LIN {X 0.073,Y -492.904,Z 865.526,A 0.000,B 0.000,C 90.000,E1 274.645} C_DIS
LIN {X -0.220,Y -493.120,Z 865.523,A 0.000,B 0.000,C 90.000,E1 274.188} C_DIS
LIN {X 0.017,Y -492.879,Z 865.520,A 0.000,B 0.000,C 90.000,E1 273.669} C_DIS
LIN {X 0.225,Y -492.231,Z 865.518,A 0.000,B 0.000,C 90.000,E1 273.154} C_DIS
LIN {X -0.033,Y -491.091,Z 865.515,A 0.000,B 0.000,C 90.000,E1 272.694} C_DIS
LIN {X 0.172,Y -489.509,Z 865.512,A 0.000,B 0.000,C 90.000,E1 272.178} C_DIS
LIN {X -0.101,Y -487.367,Z 865.509,A 0.000,B 0.000,C 90.000,E1 271.718} C_DIS
LIN {X 0.088,Y -484.709,Z 865.507,A 0.000,B 0.000,C 90.000,E1 271.203} C_DIS
LIN {X -0.225,Y -481.334,Z 865.504,A 0.000,B 0.000,C 90.000,E1 270.745} C_DIS
LIN {X -0.070,Y -477.260,Z 865.501,A 0.000,B 0.000,C 90.000,E1 270.229} C_DIS
LIN {X 0.060,Y -472.369,Z 865.498,A 0.000,B 0.000,C 90.000,E1 269.714} C_DIS
LIN {X -0.155,Y -466.565,Z 865.496,A 0.000,B 0.000,C 90.000,E1 269.255} C_DIS
LIN {X 0.090,Y -460.380,Z 865.493,A 0.000,B 0.000,C 90.000,E1 268.797} C_DIS
LIN {X -0.019,Y -457.282,Z 865.492,A 0.000,B 0.000,C 90.000,E1 268.625} C_DIS
LIN {X 0.043,Y -450.188,Z 865.490,A 0.000,B 0.000,C 90.000,E1 268.282} C_DIS
LIN {X 0.171,Y -442.949,Z 865.489,A 0.000,B 0.000,C 90.000,E1 267.993} C_DIS
LIN {X -0.152,Y -435.156,Z 865.488,A 0.000,B 0.000,C 90.000,E1 267.822} C_DIS
LIN {X -0.075,Y -427.085,Z 865.487,A 0.000,B 0.000,C 90.000,E1 267.650} C_DIS
LIN {X -0.084,Y -416.791,Z 865.486,A 0.000,B 0.000,C 90.000,E1 267.535} C_DIS
LIN {X 0.160,Y -410.055,Z 865.486,A 0.000,B 0.000,C 90.000,E1 267.478} C_DIS
LIN {X 0.053,Y -181.050,Z 865.486,A 0.000,B 0.000,C 90.000,E1 267.478} C_DIS
LIN {X -0.048,Y -180.907,Z 865.475,A 0.000,B 0.000,C 90.000,E1 265.469} C_DIS
LIN {X 0.008,Y -180.730,Z 865.470,A 0.000,B 0.000,C 90.000,E1 264.609} C_DIS
LIN {X -0.070,Y -178.819,Z 865.442,A 0.000,B 0.000,C 90.000,E1 259.567} C_DIS
LIN {X 0.012,Y -175.863,Z 865.414,A 0.000,B 0.000,C 90.000,E1 254.448} C_DIS
LIN {X 0.061,Y -173.830,Z 865.399,A 0.000,B 0.000,C 90.000,E1 251.873} C_DIS
LIN {X -0.004,Y -171.497,Z 865.380,A 0.000,B 0.000,C 90.000,E1 248.465} C_DIS
LIN {X -0.017,Y -167.726,Z 865.356,A 0.000,B 0.000,C 90.000,E1 244.152} C_DIS
LIN {X -0.001,Y -166.421,Z 865.347,A 0.000,B 0.000,C 90.000,E1 242.410} C_DIS
LIN {X -0.002,Y -163.142,Z 865.327,A 0.000,B 0.000,C 90.000,E1 238.918} C_DIS
LIN {X -0.037,Y -161.096,Z 865.313,A 0.000,B 0.000,C 90.000,E1 236.294} C_DIS
LIN {X -0.053,Y -157.825,Z 865.293,A 0.000,B 0.000,C 90.000,E1 232.763} C_DIS
LIN {X 0.010,Y -155.859,Z 865.278,A 0.000,B 0.000,C 90.000,E1 230.070} C_DIS
LIN {X 0.066,Y -152.109,Z 865.253,A 0.000,B 0.000,C 90.000,E1 225.567} C_DIS
LIN {X -0.026,Y -150.359,Z 865.238,A 0.000,B 0.000,C 90.000,E1 222.894} C_DIS
LIN {X 0.013,Y -147.095,Z 865.213,A 0.000,B 0.000,C 90.000,E1 218.338} C_DIS
LIN {X 0.008,Y -145.665,Z 865.198,A 0.000,B 0.000,C 90.000,E1 215.598} C_DIS
LIN {X 0.010,Y -143.047,Z 865.172,A 0.000,B 0.000,C 90.000,E1 211.003} C_DIS
LIN {X 0.011,Y -141.671,Z 865.152,A 0.000,B 0.000,C 90.000,E1 207.308} C_DIS
LIN {X 0.055,Y -139.452,Z 865.116,A 0.000,B 0.000,C 90.000,E1 200.791} C_DIS
LIN {X -0.023,Y -139.186,Z 865.105,A 0.000,B 0.000,C 90.000,E1 198.960} C_DIS
LIN {X -0.001,Y -138.322,Z 865.053,A 0.000,B 0.000,C 90.000,E1 189.613} C_DIS
LIN {X 0.006,Y -139.460,Z 865.007,A 0.000,B 0.000,C 90.000,E1 181.203} C_DIS
LIN {X -0.054,Y -141.016,Z 864.976,A 0.000,B 0.000,C 90.000,E1 175.641} C_DIS
LIN {X 0.037,Y -142.770,Z 864.955,A 0.000,B 0.000,C 90.000,E1 171.894} C_DIS
LIN {X -0.008,Y -145.180,Z 864.929,A 0.000,B 0.000,C 90.000,E1 167.297} C_DIS
LIN {X 0.025,Y -147.803,Z 864.909,A 0.000,B 0.000,C 90.000,E1 163.614} C_DIS
LIN {X -0.080,Y -150.489,Z 864.889,A 0.000,B 0.000,C 90.000,E1 160.007} C_DIS
LIN {X -0.007,Y -153.944,Z 864.869,A 0.000,B 0.000,C 90.000,E1 156.357} C_DIS
LIN {X 0.056,Y -157.356,Z 864.849,A 0.000,B 0.000,C 90.000,E1 152.743} C_DIS
LIN {X -0.001,Y -161.552,Z 864.829,A 0.000,B 0.000,C 90.000,E1 149.203} C_DIS
LIN {X 0.011,Y -165.749,Z 864.809,A 0.000,B 0.000,C 90.000,E1 145.674} C_DIS
LIN {X -0.002,Y -170.704,Z 864.790,A 0.000,B 0.000,C 90.000,E1 142.190} C_DIS
LIN {X -0.090,Y -175.578,Z 864.771,A 0.000,B 0.000,C 90.000,E1 138.771} C_DIS
LIN {X 0.029,Y -181.196,Z 864.752,A 0.000,B 0.000,C 90.000,E1 135.324} C_DIS
LIN {X 0.022,Y -186.657,Z 864.733,A 0.000,B 0.000,C 90.000,E1 131.962} C_DIS
LIN {X -0.034,Y -191.262,Z 864.719,A 0.000,B 0.000,C 90.000,E1 129.483} C_DIS
LIN {X -0.025,Y -193.092,Z 864.713,A 0.000,B 0.000,C 90.000,E1 128.382} C_DIS
LIN {X -0.072,Y -294.130,Z 864.713,A 0.000,B 0.000,C 90.000,E1 128.382} C_DIS
LIN {X 0.045,Y -296.837,Z 864.713,A 0.000,B 0.000,C 90.000,E1 128.302} C_DIS
LIN {X -0.152,Y -301.150,Z 864.711,A 0.000,B 0.000,C 90.000,E1 128.096} C_DIS
LIN {X 0.072,Y -303.688,Z 864.710,A 0.000,B 0.000,C 90.000,E1 127.810} C_DIS
LIN {X -0.038,Y -307.442,Z 864.707,A 0.000,B 0.000,C 90.000,E1 127.282} C_DIS
LIN {X -0.019,Y -309.008,Z 864.705,A 0.000,B 0.000,C 90.000,E1 126.950} C_DIS
LIN {X 0.186,Y -310.237,Z 864.703,A 0.000,B 0.000,C 90.000,E1 126.583} C_DIS
LIN {X -0.127,Y -321.379,Z 864.684,A 0.000,B 0.000,C 90.000,E1 123.086} C_DIS
LIN {X 0.019,Y -331.855,Z 864.668,A 0.000,B 0.000,C 90.000,E1 120.207} C_DIS
LIN {X 0.149,Y -343.684,Z 864.652,A 0.000,B 0.000,C 90.000,E1 117.385} C_DIS
LIN {X 0.142,Y -356.977,Z 864.637,A 0.000,B 0.000,C 90.000,E1 114.643} C_DIS
LIN {X -0.014,Y -370.114,Z 864.624,A 0.000,B 0.000,C 90.000,E1 112.280} C_DIS
LIN {X 0.019,Y -384.590,Z 864.611,A 0.000,B 0.000,C 90.000,E1 109.939} C_DIS
LIN {X 0.152,Y -400.512,Z 864.598,A 0.000,B 0.000,C 90.000,E1 107.638} C_DIS
LIN {X 0.055,Y -417.992,Z 864.586,A 0.000,B 0.000,C 90.000,E1 105.426} C_DIS
LIN {X -0.238,Y -437.140,Z 864.574,A 0.000,B 0.000,C 90.000,E1 103.300} C_DIS
LIN {X 0.008,Y -457.271,Z 864.562,A 0.000,B 0.000,C 90.000,E1 101.243} C_DIS
LIN {X -0.124,Y -467.492,Z 864.557,A 0.000,B 0.000,C 90.000,E1 100.310} C_DIS
LIN {X -0.128,Y -469.515,Z 864.556,A 0.000,B 0.000,C 90.000,E1 100.074} C_DIS
LIN {X -0.214,Y -471.052,Z 864.555,A 0.000,B 0.000,C 90.000,E1 99.849} C_DIS
LIN {X 0.105,Y -472.304,Z 864.553,A 0.000,B 0.000,C 90.000,E1 99.557} C_DIS
LIN {X -0.042,Y -473.223,Z 864.552,A 0.000,B 0.000,C 90.000,E1 99.321} C_DIS
LIN {X 0.070,Y -474.227,Z 864.549,A 0.000,B 0.000,C 90.000,E1 98.803} C_DIS
LIN {X 0.259,Y -474.248,Z 864.546,A 0.000,B 0.000,C 90.000,E1 98.276} C_DIS
LIN {X -0.087,Y -473.293,Z 864.543,A 0.000,B 0.000,C 90.000,E1 97.814} C_DIS
LIN {X 0.039,Y -471.201,Z 864.541,A 0.000,B 0.000,C 90.000,E1 97.296} C_DIS
LIN {X 0.195,Y -453.697,Z 864.525,A 0.000,B 0.000,C 90.000,E1 94.473} C_DIS
LIN {X -0.110,Y -443.186,Z 864.515,A 0.000,B 0.000,C 90.000,E1 92.694} C_DIS
LIN {X 0.075,Y -433.849,Z 864.506,A 0.000,B 0.000,C 90.000,E1 91.088} C_DIS
LIN {X 0.086,Y -424.216,Z 864.497,A 0.000,B 0.000,C 90.000,E1 89.484} C_DIS
LIN {X 0.030,Y -412.818,Z 864.487,A 0.000,B 0.000,C 90.000,E1 87.593} C_DIS
LIN {X 0.175,Y -401.391,Z 864.476,A 0.000,B 0.000,C 90.000,E1 85.641} C_DIS
LIN {X 0.157,Y -388.423,Z 864.463,A 0.000,B 0.000,C 90.000,E1 83.394} C_DIS
LIN {X -0.115,Y -375.665,Z 864.451,A 0.000,B 0.000,C 90.000,E1 81.141} C_DIS
LIN {X 0.130,Y -361.540,Z 864.436,A 0.000,B 0.000,C 90.000,E1 78.465} C_DIS
LIN {X -0.089,Y -350.608,Z 864.424,A 0.000,B 0.000,C 90.000,E1 76.408} C_DIS
LIN {X -0.118,Y -338.191,Z 864.411,A 0.000,B 0.000,C 90.000,E1 73.976} C_DIS
LIN {X 0.060,Y -326.043,Z 864.397,A 0.000,B 0.000,C 90.000,E1 71.456} C_DIS
LIN {X 0.064,Y -312.889,Z 864.381,A 0.000,B 0.000,C 90.000,E1 68.592} C_DIS
LIN {X -0.133,Y -302.956,Z 864.369,A 0.000,B 0.000,C 90.000,E1 66.357} C_DIS
LIN {X -0.027,Y -291.711,Z 864.354,A 0.000,B 0.000,C 90.000,E1 63.691} C_DIS
LIN {X 0.089,Y -281.990,Z 864.341,A 0.000,B 0.000,C 90.000,E1 61.307} C_DIS
LIN {X -0.042,Y -271.106,Z 864.325,A 0.000,B 0.000,C 90.000,E1 58.584} C_DIS
LIN {X 0.015,Y -258.194,Z 864.306,A 0.000,B 0.000,C 90.000,E1 55.055} C_DIS
LIN {X -0.021,Y -247.643,Z 864.288,A 0.000,B 0.000,C 90.000,E1 51.823} C_DIS
LIN {X -0.068,Y -237.007,Z 864.267,A 0.000,B 0.000,C 90.000,E1 48.162} C_DIS
LIN {X 0.017,Y -227.185,Z 864.247,A 0.000,B 0.000,C 90.000,E1 44.393} C_DIS
LIN {X 0.128,Y -218.020,Z 864.225,A 0.000,B 0.000,C 90.000,E1 40.539} C_DIS
LIN {X 0.064,Y -211.123,Z 864.208,A 0.000,B 0.000,C 90.000,E1 37.443} C_DIS
LIN {X 0.021,Y -203.152,Z 864.186,A 0.000,B 0.000,C 90.000,E1 33.499} C_DIS
LIN {X 0.075,Y -195.967,Z 864.164,A 0.000,B 0.000,C 90.000,E1 29.461} C_DIS
LIN {X -0.043,Y -190.896,Z 864.146,A 0.000,B 0.000,C 90.000,E1 26.232} C_DIS
LIN {X 0.069,Y -186.582,Z 864.127,A 0.000,B 0.000,C 90.000,E1 22.898} C_DIS
LIN {X 0.079,Y -182.215,Z 864.104,A 0.000,B 0.000,C 90.000,E1 18.725} C_DIS
LIN {X 0.014,Y -178.992,Z 864.081,A 0.000,B 0.000,C 90.000,E1 14.537} C_DIS
LIN {X -0.068,Y -176.333,Z 864.048,A 0.000,B 0.000,C 90.000,E1 8.624} C_DIS
LIN {X -0.078,Y -177.590,Z 863.974,A 0.000,B 0.000,C 90.000,E1 355.298} C_DIS
LIN {X -0.075,Y -180.602,Z 863.945,A 0.000,B 0.000,C 90.000,E1 350.208} C_DIS
LIN {X -0.059,Y -184.287,Z 863.922,A 0.000,B 0.000,C 90.000,E1 345.992} C_DIS
LIN {X -0.063,Y -189.055,Z 863.899,A 0.000,B 0.000,C 90.000,E1 341.819} C_DIS
LIN {X 0.099,Y -193.603,Z 863.880,A 0.000,B 0.000,C 90.000,E1 338.465} C_DIS
LIN {X 0.005,Y -200.178,Z 863.858,A 0.000,B 0.000,C 90.000,E1 334.409} C_DIS
LIN {X 0.014,Y -207.406,Z 863.836,A 0.000,B 0.000,C 90.000,E1 330.383} C_DIS
LIN {X 0.024,Y -215.337,Z 863.813,A 0.000,B 0.000,C 90.000,E1 326.421} C_DIS
LIN {X 0.071,Y -222.281,Z 863.796,A 0.000,B 0.000,C 90.000,E1 323.290} C_DIS
LIN {X 0.113,Y -230.938,Z 863.777,A 0.000,B 0.000,C 90.000,E1 319.828} C_DIS
LIN {X 0.083,Y -239.422,Z 863.760,A 0.000,B 0.000,C 90.000,E1 316.824} C_DIS
LIN {X 0.087,Y -248.774,Z 863.744,A 0.000,B 0.000,C 90.000,E1 313.866} C_DIS
LIN {X 0.019,Y -260.312,Z 863.726,A 0.000,B 0.000,C 90.000,E1 310.620} C_DIS
LIN {X -0.022,Y -272.802,Z 863.708,A 0.000,B 0.000,C 90.000,E1 307.443} C_DIS
LIN {X 0.013,Y -286.471,Z 863.691,A 0.000,B 0.000,C 90.000,E1 304.326} C_DIS
LIN {X -0.201,Y -301.452,Z 863.674,A 0.000,B 0.000,C 90.000,E1 301.337} C_DIS
LIN {X 0.003,Y -314.127,Z 863.661,A 0.000,B 0.000,C 90.000,E1 298.999} C_DIS
LIN {X -0.044,Y -325.947,Z 863.650,A 0.000,B 0.000,C 90.000,E1 297.078} C_DIS
LIN {X -0.044,Y -345.450,Z 863.635,A 0.000,B 0.000,C 90.000,E1 294.259} C_DIS
LIN {X 0.034,Y -369.064,Z 863.618,A 0.000,B 0.000,C 90.000,E1 291.227} C_DIS
LIN {X 0.144,Y -394.598,Z 863.602,A 0.000,B 0.000,C 90.000,E1 288.362} C_DIS
LIN {X -0.033,Y -412.830,Z 863.592,A 0.000,B 0.000,C 90.000,E1 286.496} C_DIS
LIN {X 0.054,Y -422.816,Z 863.586,A 0.000,B 0.000,C 90.000,E1 285.426} C_DIS
LIN {X 0.035,Y -432.657,Z 863.580,A 0.000,B 0.000,C 90.000,E1 284.356} C_DIS
LIN {X -0.054,Y -442.279,Z 863.574,A 0.000,B 0.000,C 90.000,E1 283.300} C_DIS
LIN {X -0.026,Y -451.331,Z 863.568,A 0.000,B 0.000,C 90.000,E1 282.243} C_DIS
LIN {X 0.119,Y -459.815,Z 863.562,A 0.000,B 0.000,C 90.000,E1 281.186} C_DIS
LIN {X -0.189,Y -467.691,Z 863.557,A 0.000,B 0.000,C 90.000,E1 280.197} C_DIS
LIN {X 0.055,Y -474.900,Z 863.551,A 0.000,B 0.000,C 90.000,E1 279.151} C_DIS
LIN {X 0.045,Y -479.741,Z 863.547,A 0.000,B 0.000,C 90.000,E1 278.398} C_DIS
LIN {X 0.073,Y -483.847,Z 863.543,A 0.000,B 0.000,C 90.000,E1 277.644} C_DIS
LIN {X -0.231,Y -486.163,Z 863.540,A 0.000,B 0.000,C 90.000,E1 277.182} C_DIS
LIN {X -0.036,Y -488.183,Z 863.537,A 0.000,B 0.000,C 90.000,E1 276.663} C_DIS
LIN {X 0.166,Y -489.862,Z 863.534,A 0.000,B 0.000,C 90.000,E1 276.144} C_DIS
LIN {X -0.109,Y -491.220,Z 863.531,A 0.000,B 0.000,C 90.000,E1 275.682} C_DIS
LIN {X 0.115,Y -492.236,Z 863.529,A 0.000,B 0.000,C 90.000,E1 275.163} C_DIS
LIN {X -0.147,Y -492.858,Z 863.526,A 0.000,B 0.000,C 90.000,E1 274.702} C_DIS
LIN {X 0.049,Y -493.070,Z 863.523,A 0.000,B 0.000,C 90.000,E1 274.188} C_DIS
LIN {X -0.205,Y -492.891,Z 863.521,A 0.000,B 0.000,C 90.000,E1 273.726} C_DIS
LIN {X 0.002,Y -492.275,Z 863.518,A 0.000,B 0.000,C 90.000,E1 273.212} C_DIS
LIN {X 0.235,Y -491.201,Z 863.515,A 0.000,B 0.000,C 90.000,E1 272.694} C_DIS
LIN {X -0.050,Y -489.671,Z 863.512,A 0.000,B 0.000,C 90.000,E1 272.236} C_DIS
LIN {X 0.166,Y -487.623,Z 863.510,A 0.000,B 0.000,C 90.000,E1 271.718} C_DIS
LIN {X -0.130,Y -484.976,Z 863.507,A 0.000,B 0.000,C 90.000,E1 271.260} C_DIS
LIN {X 0.042,Y -481.781,Z 863.504,A 0.000,B 0.000,C 90.000,E1 270.745} C_DIS
LIN {X 0.196,Y -477.767,Z 863.501,A 0.000,B 0.000,C 90.000,E1 270.229} C_DIS
LIN {X 0.024,Y -475.517,Z 863.500,A 0.000,B 0.000,C 90.000,E1 270.000} C_DIS
LIN {X 0.208,Y -470.287,Z 863.497,A 0.000,B 0.000,C 90.000,E1 269.484} C_DIS
LIN {X 0.166,Y -464.409,Z 863.495,A 0.000,B 0.000,C 90.000,E1 269.026} C_DIS
LIN {X 0.099,Y -458.056,Z 863.492,A 0.000,B 0.000,C 90.000,E1 268.625} C_DIS
LIN {X 0.104,Y -451.003,Z 863.491,A 0.000,B 0.000,C 90.000,E1 268.282} C_DIS
LIN {X 0.187,Y -443.743,Z 863.489,A 0.000,B 0.000,C 90.000,E1 267.993} C_DIS
LIN {X -0.178,Y -436.094,Z 863.488,A 0.000,B 0.000,C 90.000,E1 267.822} C_DIS
LIN {X -0.131,Y -427.988,Z 863.487,A 0.000,B 0.000,C 90.000,E1 267.650} C_DIS
LIN {X -0.133,Y -418.387,Z 863.486,A 0.000,B 0.000,C 90.000,E1 267.535} C_DIS
LIN {X 0.048,Y -410.697,Z 863.486,A 0.000,B 0.000,C 90.000,E1 267.478} C_DIS
LIN {X 0.001,Y -181.047,Z 863.486,A 0.000,B 0.000,C 90.000,E1 267.478} C_DIS
LIN {X -0.085,Y -180.906,Z 863.475,A 0.000,B 0.000,C 90.000,E1 265.469} C_DIS
LIN {X -0.028,Y -180.724,Z 863.470,A 0.000,B 0.000,C 90.000,E1 264.609} C_DIS
LIN {X 0.070,Y -178.813,Z 863.442,A 0.000,B 0.000,C 90.000,E1 259.511} C_DIS
LIN {X -0.024,Y -175.858,Z 863.414,A 0.000,B 0.000,C 90.000,E1 254.448} C_DIS
LIN {X -0.042,Y -173.186,Z 863.395,A 0.000,B 0.000,C 90.000,E1 251.040} C_DIS
LIN {X -0.040,Y -171.488,Z 863.380,A 0.000,B 0.000,C 90.000,E1 248.465} C_DIS
LIN {X -0.052,Y -167.717,Z 863.356,A 0.000,B 0.000,C 90.000,E1 244.152} C_DIS
LIN {X -0.036,Y -166.409,Z 863.347,A 0.000,B 0.000,C 90.000,E1 242.410} C_DIS
LIN {X -0.038,Y -163.132,Z 863.327,A 0.000,B 0.000,C 90.000,E1 238.918} C_DIS
LIN {X -0.071,Y -161.084,Z 863.313,A 0.000,B 0.000,C 90.000,E1 236.294} C_DIS
LIN {X 0.038,Y -157.815,Z 863.293,A 0.000,B 0.000,C 90.000,E1 232.718} C_DIS
LIN {X -0.024,Y -155.849,Z 863.278,A 0.000,B 0.000,C 90.000,E1 230.070} C_DIS
LIN {X 0.033,Y -152.099,Z 863.253,A 0.000,B 0.000,C 90.000,E1 225.567} C_DIS
LIN {X 0.051,Y -150.350,Z 863.238,A 0.000,B 0.000,C 90.000,E1 222.852} C_DIS
LIN {X -0.020,Y -147.087,Z 863.213,A 0.000,B 0.000,C 90.000,E1 218.338} C_DIS
LIN {X -0.025,Y -145.658,Z 863.198,A 0.000,B 0.000,C 90.000,E1 215.598} C_DIS
LIN {X -0.022,Y -143.040,Z 863.172,A 0.000,B 0.000,C 90.000,E1 211.003} C_DIS
LIN {X -0.021,Y -141.665,Z 863.152,A 0.000,B 0.000,C 90.000,E1 207.308} C_DIS
LIN {X 0.024,Y -139.450,Z 863.116,A 0.000,B 0.000,C 90.000,E1 200.791} C_DIS
LIN {X -0.055,Y -139.184,Z 863.105,A 0.000,B 0.000,C 90.000,E1 198.960} C_DIS
LIN {X -0.032,Y -138.321,Z 863.053,A 0.000,B 0.000,C 90.000,E1 189.613} C_DIS
LIN {X -0.025,Y -139.462,Z 863.007,A 0.000,B 0.000,C 90.000,E1 181.203} C_DIS
LIN {X 0.055,Y -141.021,Z 862.976,A 0.000,B 0.000,C 90.000,E1 175.584} C_DIS
LIN {X 0.010,Y -142.386,Z 862.960,A 0.000,B 0.000,C 90.000,E1 172.818} C_DIS
LIN {X -0.069,Y -144.616,Z 862.934,A 0.000,B 0.000,C 90.000,E1 168.229} C_DIS
LIN {X -0.008,Y -147.811,Z 862.909,A 0.000,B 0.000,C 90.000,E1 163.614} C_DIS
LIN {X 0.079,Y -150.499,Z 862.889,A 0.000,B 0.000,C 90.000,E1 159.934} C_DIS
LIN {X -0.041,Y -153.957,Z 862.869,A 0.000,B 0.000,C 90.000,E1 156.357} C_DIS
LIN {X 0.021,Y -157.369,Z 862.849,A 0.000,B 0.000,C 90.000,E1 152.743} C_DIS
LIN {X -0.035,Y -161.568,Z 862.829,A 0.000,B 0.000,C 90.000,E1 149.203} C_DIS
LIN {X -0.023,Y -165.766,Z 862.809,A 0.000,B 0.000,C 90.000,E1 145.674} C_DIS
LIN {X -0.038,Y -170.723,Z 862.790,A 0.000,B 0.000,C 90.000,E1 142.190} C_DIS
LIN {X 0.005,Y -175.596,Z 862.771,A 0.000,B 0.000,C 90.000,E1 138.728} C_DIS
LIN {X -0.008,Y -181.213,Z 862.752,A 0.000,B 0.000,C 90.000,E1 135.324} C_DIS
LIN {X -0.016,Y -186.678,Z 862.733,A 0.000,B 0.000,C 90.000,E1 131.962} C_DIS
LIN {X -0.073,Y -191.280,Z 862.719,A 0.000,B 0.000,C 90.000,E1 129.483} C_DIS
LIN {X 0.001,Y -193.078,Z 862.713,A 0.000,B 0.000,C 90.000,E1 128.382} C_DIS
LIN {X -0.047,Y -294.510,Z 862.713,A 0.000,B 0.000,C 90.000,E1 128.382} C_DIS
LIN {X -0.043,Y -300.960,Z 862.712,A 0.000,B 0.000,C 90.000,E1 128.096} C_DIS
LIN {X 0.012,Y -303.823,Z 862.710,A 0.000,B 0.000,C 90.000,E1 127.810} C_DIS
LIN {X 0.136,Y -307.514,Z 862.707,A 0.000,B 0.000,C 90.000,E1 127.237} C_DIS
LIN {X -0.089,Y -309.054,Z 862.705,A 0.000,B 0.000,C 90.000,E1 126.950} C_DIS
LIN {X 0.117,Y -310.262,Z 862.703,A 0.000,B 0.000,C 90.000,E1 126.583} C_DIS
LIN {X 0.070,Y -321.402,Z 862.684,A 0.000,B 0.000,C 90.000,E1 123.038} C_DIS
LIN {X -0.054,Y -331.884,Z 862.668,A 0.000,B 0.000,C 90.000,E1 120.207} C_DIS
LIN {X 0.075,Y -343.719,Z 862.652,A 0.000,B 0.000,C 90.000,E1 117.385} C_DIS
LIN {X 0.065,Y -357.018,Z 862.637,A 0.000,B 0.000,C 90.000,E1 114.643} C_DIS
LIN {X -0.092,Y -370.160,Z 862.624,A 0.000,B 0.000,C 90.000,E1 112.280} C_DIS
LIN {X -0.061,Y -384.644,Z 862.611,A 0.000,B 0.000,C 90.000,E1 109.939} C_DIS
LIN {X 0.070,Y -400.573,Z 862.598,A 0.000,B 0.000,C 90.000,E1 107.638} C_DIS
LIN {X -0.029,Y -418.061,Z 862.586,A 0.000,B 0.000,C 90.000,E1 105.426} C_DIS
LIN {X 0.101,Y -437.217,Z 862.574,A 0.000,B 0.000,C 90.000,E1 103.244} C_DIS
LIN {X -0.074,Y -457.352,Z 862.562,A 0.000,B 0.000,C 90.000,E1 101.243} C_DIS
LIN {X -0.205,Y -467.566,Z 862.557,A 0.000,B 0.000,C 90.000,E1 100.310} C_DIS
LIN {X 0.249,Y -469.577,Z 862.556,A 0.000,B 0.000,C 90.000,E1 100.018} C_DIS
LIN {X 0.162,Y -471.105,Z 862.555,A 0.000,B 0.000,C 90.000,E1 99.792} C_DIS
LIN {X 0.017,Y -472.348,Z 862.553,A 0.000,B 0.000,C 90.000,E1 99.557} C_DIS
LIN {X -0.131,Y -473.260,Z 862.552,A 0.000,B 0.000,C 90.000,E1 99.321} C_DIS
LIN {X -0.019,Y -474.251,Z 862.549,A 0.000,B 0.000,C 90.000,E1 98.803} C_DIS
LIN {X 0.170,Y -474.260,Z 862.546,A 0.000,B 0.000,C 90.000,E1 98.276} C_DIS
LIN {X -0.174,Y -473.293,Z 862.543,A 0.000,B 0.000,C 90.000,E1 97.814} C_DIS
LIN {X -0.048,Y -471.186,Z 862.541,A 0.000,B 0.000,C 90.000,E1 97.296} C_DIS
LIN {X 0.110,Y -453.659,Z 862.525,A 0.000,B 0.000,C 90.000,E1 94.473} C_DIS
LIN {X -0.193,Y -443.139,Z 862.515,A 0.000,B 0.000,C 90.000,E1 92.694} C_DIS
LIN {X -0.172,Y -435.409,Z 862.508,A 0.000,B 0.000,C 90.000,E1 91.375} C_DIS
LIN {X -0.131,Y -425.792,Z 862.499,A 0.000,B 0.000,C 90.000,E1 89.771} C_DIS
LIN {X -0.141,Y -414.402,Z 862.488,A 0.000,B 0.000,C 90.000,E1 87.879} C_DIS
LIN {X 0.039,Y -402.966,Z 862.477,A 0.000,B 0.000,C 90.000,E1 85.927} C_DIS
LIN {X 0.026,Y -389.955,Z 862.465,A 0.000,B 0.000,C 90.000,E1 83.685} C_DIS
LIN {X 0.162,Y -377.183,Z 862.452,A 0.000,B 0.000,C 90.000,E1 81.376} C_DIS
LIN {X 0.082,Y -363.049,Z 862.438,A 0.000,B 0.000,C 90.000,E1 78.757} C_DIS
LIN {X -0.108,Y -352.142,Z 862.426,A 0.000,B 0.000,C 90.000,E1 76.700} C_DIS
LIN {X -0.096,Y -339.756,Z 862.412,A 0.000,B 0.000,C 90.000,E1 74.267} C_DIS
LIN {X 0.024,Y -327.552,Z 862.399,A 0.000,B 0.000,C 90.000,E1 71.764} C_DIS
LIN {X 0.072,Y -314.371,Z 862.383,A 0.000,B 0.000,C 90.000,E1 68.901} C_DIS
LIN {X -0.099,Y -304.431,Z 862.370,A 0.000,B 0.000,C 90.000,E1 66.666} C_DIS
LIN {X -0.082,Y -293.219,Z 862.356,A 0.000,B 0.000,C 90.000,E1 64.024} C_DIS
LIN {X 0.068,Y -283.543,Z 862.343,A 0.000,B 0.000,C 90.000,E1 61.641} C_DIS
LIN {X -0.026,Y -272.640,Z 862.327,A 0.000,B 0.000,C 90.000,E1 58.918} C_DIS
LIN {X 0.081,Y -259.711,Z 862.308,A 0.000,B 0.000,C 90.000,E1 55.388} C_DIS
LIN {X -0.066,Y -249.084,Z 862.290,A 0.000,B 0.000,C 90.000,E1 52.190} C_DIS
LIN {X 0.124,Y -239.384,Z 862.272,A 0.000,B 0.000,C 90.000,E1 48.852} C_DIS
LIN {X -0.044,Y -229.411,Z 862.251,A 0.000,B 0.000,C 90.000,E1 45.162} C_DIS
LIN {X -0.033,Y -220.147,Z 862.230,A 0.000,B 0.000,C 90.000,E1 41.353} C_DIS
LIN {X -0.042,Y -213.109,Z 862.212,A 0.000,B 0.000,C 90.000,E1 38.257} C_DIS
LIN {X -0.014,Y -206.594,Z 862.195,A 0.000,B 0.000,C 90.000,E1 35.105} C_DIS
LIN {X -0.052,Y -200.507,Z 862.177,A 0.000,B 0.000,C 90.000,E1 31.926} C_DIS
LIN {X -0.043,Y -194.951,Z 862.159,A 0.000,B 0.000,C 90.000,E1 28.693} C_DIS
LIN {X -0.008,Y -190.026,Z 862.141,A 0.000,B 0.000,C 90.000,E1 25.412} C_DIS
LIN {X 0.081,Y -185.895,Z 862.123,A 0.000,B 0.000,C 90.000,E1 22.078} C_DIS
LIN {X -0.057,Y -181.800,Z 862.100,A 0.000,B 0.000,C 90.000,E1 17.946} C_DIS
LIN {X -0.004,Y -178.803,Z 862.076,A 0.000,B 0.000,C 90.000,E1 13.716} C_DIS
LIN {X 0.053,Y -176.436,Z 862.043,A 0.000,B 0.000,C 90.000,E1 7.757} C_DIS
LIN {X 0.074,Y -177.588,Z 861.978,A 0.000,B 0.000,C 90.000,E1 356.102} C_DIS
LIN {X 0.030,Y -180.367,Z 861.950,A 0.000,B 0.000,C 90.000,E1 351.027} C_DIS
LIN {X -0.007,Y -183.835,Z 861.927,A 0.000,B 0.000,C 90.000,E1 346.825} C_DIS
LIN {X -0.027,Y -188.393,Z 861.904,A 0.000,B 0.000,C 90.000,E1 342.653} C_DIS
LIN {X -0.009,Y -192.767,Z 861.885,A 0.000,B 0.000,C 90.000,E1 339.337} C_DIS
LIN {X 0.024,Y -197.799,Z 861.867,A 0.000,B 0.000,C 90.000,E1 336.049} C_DIS
LIN {X -0.050,Y -204.748,Z 861.844,A 0.000,B 0.000,C 90.000,E1 332.025} C_DIS
LIN {X -0.002,Y -210.779,Z 861.827,A 0.000,B 0.000,C 90.000,E1 328.820} C_DIS
LIN {X -0.022,Y -218.984,Z 861.805,A 0.000,B 0.000,C 90.000,E1 324.895} C_DIS
LIN {X -0.113,Y -226.268,Z 861.788,A 0.000,B 0.000,C 90.000,E1 321.823} C_DIS
LIN {X 0.028,Y -235.321,Z 861.769,A 0.000,B 0.000,C 90.000,E1 318.366} C_DIS
LIN {X 0.086,Y -245.347,Z 861.750,A 0.000,B 0.000,C 90.000,E1 315.000} C_DIS
LIN {X -0.092,Y -256.543,Z 861.732,A 0.000,B 0.000,C 90.000,E1 311.757} C_DIS
LIN {X -0.084,Y -268.637,Z 861.714,A 0.000,B 0.000,C 90.000,E1 308.543} C_DIS
LIN {X 0.000,Y -281.849,Z 861.697,A 0.000,B 0.000,C 90.000,E1 305.391} C_DIS
LIN {X -0.026,Y -296.316,Z 861.680,A 0.000,B 0.000,C 90.000,E1 302.339} C_DIS
LIN {X 0.149,Y -312.152,Z 861.663,A 0.000,B 0.000,C 90.000,E1 299.333} C_DIS
LIN {X -0.138,Y -325.795,Z 861.651,A 0.000,B 0.000,C 90.000,E1 297.129} C_DIS
LIN {X 0.159,Y -345.209,Z 861.635,A 0.000,B 0.000,C 90.000,E1 294.259} C_DIS
LIN {X -0.119,Y -366.157,Z 861.620,A 0.000,B 0.000,C 90.000,E1 291.589} C_DIS
LIN {X -0.014,Y -394.129,Z 861.602,A 0.000,B 0.000,C 90.000,E1 288.417} C_DIS
LIN {X 0.138,Y -412.416,Z 861.592,A 0.000,B 0.000,C 90.000,E1 286.496} C_DIS
LIN {X 0.206,Y -422.440,Z 861.586,A 0.000,B 0.000,C 90.000,E1 285.426} C_DIS
LIN {X 0.180,Y -432.327,Z 861.580,A 0.000,B 0.000,C 90.000,E1 284.356} C_DIS
LIN {X 0.091,Y -441.966,Z 861.574,A 0.000,B 0.000,C 90.000,E1 283.300} C_DIS
LIN {X 0.118,Y -451.066,Z 861.568,A 0.000,B 0.000,C 90.000,E1 282.243} C_DIS
LIN {X -0.197,Y -459.556,Z 861.562,A 0.000,B 0.000,C 90.000,E1 281.243} C_DIS
LIN {X -0.056,Y -467.473,Z 861.557,A 0.000,B 0.000,C 90.000,E1 280.197} C_DIS
LIN {X 0.188,Y -474.720,Z 861.551,A 0.000,B 0.000,C 90.000,E1 279.151} C_DIS
LIN {X 0.179,Y -479.552,Z 861.547,A 0.000,B 0.000,C 90.000,E1 278.398} C_DIS
LIN {X 0.205,Y -483.677,Z 861.543,A 0.000,B 0.000,C 90.000,E1 277.644} C_DIS
LIN {X -0.097,Y -486.026,Z 861.540,A 0.000,B 0.000,C 90.000,E1 277.182} C_DIS
LIN {X 0.096,Y -488.061,Z 861.537,A 0.000,B 0.000,C 90.000,E1 276.663} C_DIS
LIN {X -0.190,Y -489.745,Z 861.534,A 0.000,B 0.000,C 90.000,E1 276.201} C_DIS
LIN {X 0.023,Y -491.159,Z 861.532,A 0.000,B 0.000,C 90.000,E1 275.682} C_DIS
LIN {X 0.246,Y -492.167,Z 861.529,A 0.000,B 0.000,C 90.000,E1 275.163} C_DIS
LIN {X -0.016,Y -492.799,Z 861.526,A 0.000,B 0.000,C 90.000,E1 274.702} C_DIS
LIN {X 0.180,Y -493.046,Z 861.523,A 0.000,B 0.000,C 90.000,E1 274.188} C_DIS
LIN {X -0.075,Y -492.879,Z 861.521,A 0.000,B 0.000,C 90.000,E1 273.726} C_DIS
LIN {X 0.132,Y -492.323,Z 861.518,A 0.000,B 0.000,C 90.000,E1 273.212} C_DIS
LIN {X -0.126,Y -491.295,Z 861.515,A 0.000,B 0.000,C 90.000,E1 272.751} C_DIS
LIN {X 0.080,Y -489.807,Z 861.512,A 0.000,B 0.000,C 90.000,E1 272.236} C_DIS
LIN {X -0.192,Y -487.799,Z 861.510,A 0.000,B 0.000,C 90.000,E1 271.776} C_DIS
LIN {X -0.001,Y -485.250,Z 861.507,A 0.000,B 0.000,C 90.000,E1 271.260} C_DIS
LIN {X 0.172,Y -482.054,Z 861.504,A 0.000,B 0.000,C 90.000,E1 270.745} C_DIS
LIN {X -0.152,Y -478.143,Z 861.501,A 0.000,B 0.000,C 90.000,E1 270.286} C_DIS
LIN {X -0.015,Y -473.460,Z 861.499,A 0.000,B 0.000,C 90.000,E1 269.771} C_DIS
LIN {X 0.101,Y -467.743,Z 861.496,A 0.000,B 0.000,C 90.000,E1 269.255} C_DIS
LIN {X 0.206,Y -461.527,Z 861.493,A 0.000,B 0.000,C 90.000,E1 268.797} C_DIS
LIN {X 0.054,Y -458.437,Z 861.492,A 0.000,B 0.000,C 90.000,E1 268.625} C_DIS
LIN {X -0.094,Y -454.832,Z 861.491,A 0.000,B 0.000,C 90.000,E1 268.453} C_DIS
LIN {X 0.171,Y -447.614,Z 861.490,A 0.000,B 0.000,C 90.000,E1 268.108} C_DIS
LIN {X -0.017,Y -439.995,Z 861.488,A 0.000,B 0.000,C 90.000,E1 267.879} C_DIS
LIN {X -0.197,Y -431.744,Z 861.487,A 0.000,B 0.000,C 90.000,E1 267.707} C_DIS
LIN {X 0.050,Y -423.117,Z 861.486,A 0.000,B 0.000,C 90.000,E1 267.535} C_DIS
LIN {X -0.086,Y -412.785,Z 861.486,A 0.000,B 0.000,C 90.000,E1 267.478} C_DIS
LIN {X -0.056,Y -181.045,Z 861.486,A 0.000,B 0.000,C 90.000,E1 267.478} C_DIS
LIN {X 0.042,Y -180.906,Z 861.475,A 0.000,B 0.000,C 90.000,E1 265.412} C_DIS
LIN {X -0.082,Y -180.716,Z 861.470,A 0.000,B 0.000,C 90.000,E1 264.609} C_DIS
LIN {X 0.016,Y -178.803,Z 861.442,A 0.000,B 0.000,C 90.000,E1 259.511} C_DIS
LIN {X 0.093,Y -175.848,Z 861.413,A 0.000,B 0.000,C 90.000,E1 254.393} C_DIS
LIN {X 0.052,Y -172.584,Z 861.390,A 0.000,B 0.000,C 90.000,E1 250.134} C_DIS
LIN {X 0.068,Y -171.473,Z 861.380,A 0.000,B 0.000,C 90.000,E1 248.411} C_DIS
LIN {X 0.048,Y -167.704,Z 861.356,A 0.000,B 0.000,C 90.000,E1 244.101} C_DIS
LIN {X 0.061,Y -166.391,Z 861.347,A 0.000,B 0.000,C 90.000,E1 242.359} C_DIS
LIN {X 0.052,Y -163.118,Z 861.327,A 0.000,B 0.000,C 90.000,E1 238.869} C_DIS
LIN {X 0.102,Y -161.067,Z 861.313,A 0.000,B 0.000,C 90.000,E1 236.215} C_DIS
LIN {X -0.011,Y -157.800,Z 861.293,A 0.000,B 0.000,C 90.000,E1 232.718} C_DIS
LIN {X -0.073,Y -155.837,Z 861.278,A 0.000,B 0.000,C 90.000,E1 230.070} C_DIS
LIN {X -0.016,Y -152.087,Z 861.253,A 0.000,B 0.000,C 90.000,E1 225.567} C_DIS
LIN {X 0.003,Y -150.337,Z 861.238,A 0.000,B 0.000,C 90.000,E1 222.852} C_DIS
LIN {X 0.024,Y -147.077,Z 861.213,A 0.000,B 0.000,C 90.000,E1 218.302} C_DIS
LIN {X -0.072,Y -145.651,Z 861.198,A 0.000,B 0.000,C 90.000,E1 215.598} C_DIS
LIN {X -0.068,Y -143.032,Z 861.172,A 0.000,B 0.000,C 90.000,E1 211.003} C_DIS
LIN {X 0.059,Y -141.657,Z 861.152,A 0.000,B 0.000,C 90.000,E1 207.257} C_DIS
LIN {X -0.022,Y -139.447,Z 861.115,A 0.000,B 0.000,C 90.000,E1 200.791} C_DIS
LIN {X 0.031,Y -139.180,Z 861.105,A 0.000,B 0.000,C 90.000,E1 198.906} C_DIS
LIN {X 0.059,Y -138.320,Z 861.053,A 0.000,B 0.000,C 90.000,E1 189.557} C_DIS
LIN {X 0.068,Y -139.465,Z 861.007,A 0.000,B 0.000,C 90.000,E1 181.146} C_DIS
LIN {X 0.010,Y -141.029,Z 860.975,A 0.000,B 0.000,C 90.000,E1 175.584} C_DIS
LIN {X -0.036,Y -142.396,Z 860.960,A 0.000,B 0.000,C 90.000,E1 172.818} C_DIS
LIN {X 0.026,Y -144.628,Z 860.934,A 0.000,B 0.000,C 90.000,E1 168.173} C_DIS
LIN {X -0.056,Y -147.823,Z 860.909,A 0.000,B 0.000,C 90.000,E1 163.614} C_DIS
LIN {X 0.031,Y -150.514,Z 860.889,A 0.000,B 0.000,C 90.000,E1 159.934} C_DIS
LIN {X 0.052,Y -153.976,Z 860.868,A 0.000,B 0.000,C 90.000,E1 156.305} C_DIS
LIN {X -0.028,Y -157.388,Z 860.849,A 0.000,B 0.000,C 90.000,E1 152.743} C_DIS
LIN {X -0.086,Y -161.591,Z 860.829,A 0.000,B 0.000,C 90.000,E1 149.203} C_DIS
LIN {X -0.075,Y -165.788,Z 860.809,A 0.000,B 0.000,C 90.000,E1 145.674} C_DIS
LIN {X -0.090,Y -170.751,Z 860.790,A 0.000,B 0.000,C 90.000,E1 142.190} C_DIS
LIN {X 0.068,Y -175.623,Z 860.771,A 0.000,B 0.000,C 90.000,E1 138.690} C_DIS
LIN {X -0.062,Y -181.238,Z 860.752,A 0.000,B 0.000,C 90.000,E1 135.324} C_DIS
LIN {X 0.068,Y -186.708,Z 860.733,A 0.000,B 0.000,C 90.000,E1 131.919} C_DIS
LIN {X 0.020,Y -191.308,Z 860.719,A 0.000,B 0.000,C 90.000,E1 129.439} C_DIS
LIN {X 0.034,Y -193.062,Z 860.713,A 0.000,B 0.000,C 90.000,E1 128.382} C_DIS
LIN {X 0.016,Y -294.363,Z 860.713,A 0.000,B 0.000,C 90.000,E1 128.382} C_DIS
LIN {X 0.052,Y -296.229,Z 860.713,A 0.000,B 0.000,C 90.000,E1 128.338} C_DIS
LIN {X -0.130,Y -301.247,Z 860.711,A 0.000,B 0.000,C 90.000,E1 128.096} C_DIS
LIN {X -0.076,Y -304.003,Z 860.710,A 0.000,B 0.000,C 90.000,E1 127.810} C_DIS
LIN {X -0.043,Y -307.692,Z 860.707,A 0.000,B 0.000,C 90.000,E1 127.237} C_DIS
LIN {X 0.164,Y -309.182,Z 860.705,A 0.000,B 0.000,C 90.000,E1 126.870} C_DIS
LIN {X -0.064,Y -310.351,Z 860.703,A 0.000,B 0.000,C 90.000,E1 126.583} C_DIS
LIN {X -0.192,Y -320.407,Z 860.685,A 0.000,B 0.000,C 90.000,E1 123.372} C_DIS
LIN {X 0.101,Y -330.756,Z 860.669,A 0.000,B 0.000,C 90.000,E1 120.463} C_DIS
LIN {X 0.195,Y -342.453,Z 860.654,A 0.000,B 0.000,C 90.000,E1 117.641} C_DIS
LIN {X 0.158,Y -355.599,Z 860.638,A 0.000,B 0.000,C 90.000,E1 114.899} C_DIS
LIN {X 0.113,Y -368.597,Z 860.625,A 0.000,B 0.000,C 90.000,E1 112.514} C_DIS
LIN {X 0.104,Y -382.924,Z 860.612,A 0.000,B 0.000,C 90.000,E1 110.174} C_DIS
LIN {X 0.192,Y -398.685,Z 860.599,A 0.000,B 0.000,C 90.000,E1 107.873} C_DIS
LIN {X 0.048,Y -415.992,Z 860.587,A 0.000,B 0.000,C 90.000,E1 105.662} C_DIS
LIN {X 0.123,Y -434.958,Z 860.575,A 0.000,B 0.000,C 90.000,E1 103.480} C_DIS
LIN {X -0.208,Y -455.027,Z 860.564,A 0.000,B 0.000,C 90.000,E1 101.478} C_DIS
LIN {X 0.056,Y -467.780,Z 860.557,A 0.000,B 0.000,C 90.000,E1 100.254} C_DIS
LIN {X 0.038,Y -469.754,Z 860.556,A 0.000,B 0.000,C 90.000,E1 100.018} C_DIS
LIN {X -0.061,Y -471.255,Z 860.554,A 0.000,B 0.000,C 90.000,E1 99.792} C_DIS
LIN {X -0.207,Y -472.466,Z 860.553,A 0.000,B 0.000,C 90.000,E1 99.557} C_DIS
LIN {X 0.112,Y -473.351,Z 860.552,A 0.000,B 0.000,C 90.000,E1 99.265} C_DIS
LIN {X -0.243,Y -474.298,Z 860.549,A 0.000,B 0.000,C 90.000,E1 98.803} C_DIS
LIN {X -0.053,Y -474.265,Z 860.546,A 0.000,B 0.000,C 90.000,E1 98.276} C_DIS
LIN {X 0.071,Y -473.253,Z 860.543,A 0.000,B 0.000,C 90.000,E1 97.757} C_DIS
LIN {X -0.130,Y -472.334,Z 860.542,A 0.000,B 0.000,C 90.000,E1 97.530} C_DIS
LIN {X 0.198,Y -471.088,Z 860.540,A 0.000,B 0.000,C 90.000,E1 97.239} C_DIS
LIN {X -0.112,Y -453.517,Z 860.525,A 0.000,B 0.000,C 90.000,E1 94.473} C_DIS
LIN {X 0.029,Y -442.994,Z 860.515,A 0.000,B 0.000,C 90.000,E1 92.636} C_DIS
LIN {X 0.046,Y -435.257,Z 860.507,A 0.000,B 0.000,C 90.000,E1 91.318} C_DIS
LIN {X 0.079,Y -425.638,Z 860.498,A 0.000,B 0.000,C 90.000,E1 89.714} C_DIS
LIN {X 0.060,Y -414.246,Z 860.488,A 0.000,B 0.000,C 90.000,E1 87.822} C_DIS
LIN {X -0.170,Y -402.808,Z 860.477,A 0.000,B 0.000,C 90.000,E1 85.927} C_DIS
LIN {X -0.180,Y -389.789,Z 860.465,A 0.000,B 0.000,C 90.000,E1 83.685} C_DIS
LIN {X -0.042,Y -377.019,Z 860.452,A 0.000,B 0.000,C 90.000,E1 81.376} C_DIS
LIN {X -0.118,Y -362.896,Z 860.437,A 0.000,B 0.000,C 90.000,E1 78.757} C_DIS
LIN {X 0.036,Y -352.035,Z 860.426,A 0.000,B 0.000,C 90.000,E1 76.645} C_DIS
LIN {X 0.041,Y -341.203,Z 860.414,A 0.000,B 0.000,C 90.000,E1 74.519} C_DIS
LIN {X -0.031,Y -328.998,Z 860.400,A 0.000,B 0.000,C 90.000,E1 72.054} C_DIS
LIN {X -0.046,Y -315.766,Z 860.384,A 0.000,B 0.000,C 90.000,E1 69.209} C_DIS
LIN {X 0.004,Y -304.408,Z 860.370,A 0.000,B 0.000,C 90.000,E1 66.613} C_DIS
LIN {X 0.011,Y -293.234,Z 860.355,A 0.000,B 0.000,C 90.000,E1 63.973} C_DIS
LIN {X -0.096,Y -283.610,Z 860.342,A 0.000,B 0.000,C 90.000,E1 61.641} C_DIS
LIN {X 0.051,Y -272.742,Z 860.327,A 0.000,B 0.000,C 90.000,E1 58.869} C_DIS
LIN {X -0.065,Y -259.912,Z 860.308,A 0.000,B 0.000,C 90.000,E1 55.388} C_DIS
LIN {X 0.016,Y -248.203,Z 860.288,A 0.000,B 0.000,C 90.000,E1 51.778} C_DIS
LIN {X 0.133,Y -237.588,Z 860.267,A 0.000,B 0.000,C 90.000,E1 48.081} C_DIS
LIN {X 0.068,Y -227.781,Z 860.247,A 0.000,B 0.000,C 90.000,E1 44.352} C_DIS
LIN {X 0.039,Y -218.643,Z 860.225,A 0.000,B 0.000,C 90.000,E1 40.539} C_DIS
LIN {X -0.006,Y -211.721,Z 860.208,A 0.000,B 0.000,C 90.000,E1 37.443} C_DIS
LIN {X 0.032,Y -205.299,Z 860.190,A 0.000,B 0.000,C 90.000,E1 34.278} C_DIS
LIN {X 0.025,Y -199.321,Z 860.173,A 0.000,B 0.000,C 90.000,E1 31.082} C_DIS
LIN {X 0.008,Y -193.918,Z 860.155,A 0.000,B 0.000,C 90.000,E1 27.847} C_DIS
LIN {X -0.066,Y -189.180,Z 860.136,A 0.000,B 0.000,C 90.000,E1 24.591} C_DIS
LIN {X -0.071,Y -185.229,Z 860.118,A 0.000,B 0.000,C 90.000,E1 21.280} C_DIS
LIN {X -0.054,Y -181.390,Z 860.095,A 0.000,B 0.000,C 90.000,E1 17.094} C_DIS
LIN {X 0.025,Y -178.205,Z 860.067,A 0.000,B 0.000,C 90.000,E1 12.007} C_DIS
LIN {X 0.050,Y -176.311,Z 860.020,A 0.000,B 0.000,C 90.000,E1 3.498} C_DIS
LIN {X -0.059,Y -178.302,Z 859.974,A 0.000,B 0.000,C 90.000,E1 355.298} C_DIS
LIN {X -0.028,Y -181.346,Z 859.946,A 0.000,B 0.000,C 90.000,E1 350.208} C_DIS
LIN {X 0.011,Y -185.045,Z 859.922,A 0.000,B 0.000,C 90.000,E1 345.992} C_DIS
LIN {X 0.033,Y -189.803,Z 859.899,A 0.000,B 0.000,C 90.000,E1 341.819} C_DIS
LIN {X -0.036,Y -194.317,Z 859.881,A 0.000,B 0.000,C 90.000,E1 338.539} C_DIS
LIN {X -0.032,Y -200.818,Z 859.858,A 0.000,B 0.000,C 90.000,E1 334.460} C_DIS
LIN {X -0.102,Y -207.978,Z 859.836,A 0.000,B 0.000,C 90.000,E1 330.461} C_DIS
LIN {X -0.083,Y -215.885,Z 859.814,A 0.000,B 0.000,C 90.000,E1 326.501} C_DIS
LIN {X 0.105,Y -222.790,Z 859.796,A 0.000,B 0.000,C 90.000,E1 323.336} C_DIS
LIN {X 0.026,Y -231.438,Z 859.777,A 0.000,B 0.000,C 90.000,E1 319.908} C_DIS
LIN {X -0.023,Y -240.984,Z 859.759,A 0.000,B 0.000,C 90.000,E1 316.539} C_DIS
LIN {X 0.013,Y -251.605,Z 859.740,A 0.000,B 0.000,C 90.000,E1 313.218} C_DIS
LIN {X 0.050,Y -263.269,Z 859.722,A 0.000,B 0.000,C 90.000,E1 309.967} C_DIS
LIN {X 0.097,Y -275.922,Z 859.705,A 0.000,B 0.000,C 90.000,E1 306.790} C_DIS
LIN {X 0.062,Y -289.737,Z 859.687,A 0.000,B 0.000,C 90.000,E1 303.706} C_DIS
LIN {X -0.057,Y -304.868,Z 859.671,A 0.000,B 0.000,C 90.000,E1 300.718} C_DIS
LIN {X -0.081,Y -317.743,Z 859.658,A 0.000,B 0.000,C 90.000,E1 298.437} C_DIS
LIN {X 0.096,Y -329.788,Z 859.647,A 0.000,B 0.000,C 90.000,E1 296.488} C_DIS
LIN {X 0.063,Y -349.421,Z 859.632,A 0.000,B 0.000,C 90.000,E1 293.695} C_DIS
LIN {X 0.086,Y -368.301,Z 859.618,A 0.000,B 0.000,C 90.000,E1 291.280} C_DIS
LIN {X 0.038,Y -393.909,Z 859.602,A 0.000,B 0.000,C 90.000,E1 288.417} C_DIS
LIN {X -0.087,Y -411.990,Z 859.592,A 0.000,B 0.000,C 90.000,E1 286.551} C_DIS
LIN {X 0.104,Y -424.613,Z 859.584,A 0.000,B 0.000,C 90.000,E1 285.190} C_DIS
LIN {X 0.051,Y -434.477,Z 859.578,A 0.000,B 0.000,C 90.000,E1 284.120} C_DIS
LIN {X -0.015,Y -444.028,Z 859.573,A 0.000,B 0.000,C 90.000,E1 283.063} C_DIS
LIN {X 0.033,Y -452.963,Z 859.567,A 0.000,B 0.000,C 90.000,E1 282.007} C_DIS
LIN {X 0.188,Y -461.375,Z 859.561,A 0.000,B 0.000,C 90.000,E1 280.950} C_DIS
LIN {X -0.104,Y -469.137,Z 859.555,A 0.000,B 0.000,C 90.000,E1 279.962} C_DIS
LIN {X 0.156,Y -476.223,Z 859.550,A 0.000,B 0.000,C 90.000,E1 278.916} C_DIS
LIN {X 0.152,Y -480.858,Z 859.545,A 0.000,B 0.000,C 90.000,E1 278.163} C_DIS
LIN {X 0.191,Y -484.782,Z 859.541,A 0.000,B 0.000,C 90.000,E1 277.409} C_DIS
LIN {X 0.201,Y -487.933,Z 859.537,A 0.000,B 0.000,C 90.000,E1 276.663} C_DIS
LIN {X -0.084,Y -489.645,Z 859.534,A 0.000,B 0.000,C 90.000,E1 276.201} C_DIS
LIN {X 0.128,Y -491.049,Z 859.532,A 0.000,B 0.000,C 90.000,E1 275.682} C_DIS
LIN {X -0.140,Y -492.101,Z 859.529,A 0.000,B 0.000,C 90.000,E1 275.220} C_DIS
LIN {X 0.088,Y -492.745,Z 859.526,A 0.000,B 0.000,C 90.000,E1 274.702} C_DIS
LIN {X -0.208,Y -493.020,Z 859.523,A 0.000,B 0.000,C 90.000,E1 274.245} C_DIS
LIN {X 0.028,Y -492.891,Z 859.521,A 0.000,B 0.000,C 90.000,E1 273.726} C_DIS
LIN {X -0.257,Y -492.335,Z 859.518,A 0.000,B 0.000,C 90.000,E1 273.269} C_DIS
LIN {X -0.023,Y -491.352,Z 859.515,A 0.000,B 0.000,C 90.000,E1 272.751} C_DIS
LIN {X 0.182,Y -489.890,Z 859.513,A 0.000,B 0.000,C 90.000,E1 272.236} C_DIS
LIN {X -0.089,Y -487.958,Z 859.510,A 0.000,B 0.000,C 90.000,E1 271.776} C_DIS
LIN {X 0.102,Y -485.443,Z 859.507,A 0.000,B 0.000,C 90.000,E1 271.260} C_DIS
LIN {X -0.208,Y -482.282,Z 859.504,A 0.000,B 0.000,C 90.000,E1 270.802} C_DIS
LIN {X -0.049,Y -478.433,Z 859.502,A 0.000,B 0.000,C 90.000,E1 270.286} C_DIS
LIN {X 0.088,Y -473.857,Z 859.499,A 0.000,B 0.000,C 90.000,E1 269.771} C_DIS
LIN {X 0.198,Y -468.203,Z 859.496,A 0.000,B 0.000,C 90.000,E1 269.255} C_DIS
LIN {X -0.163,Y -462.139,Z 859.494,A 0.000,B 0.000,C 90.000,E1 268.854} C_DIS
LIN {X -0.078,Y -455.418,Z 859.491,A 0.000,B 0.000,C 90.000,E1 268.453} C_DIS
LIN {X 0.117,Y -448.111,Z 859.490,A 0.000,B 0.000,C 90.000,E1 268.108} C_DIS
LIN {X -0.081,Y -440.539,Z 859.488,A 0.000,B 0.000,C 90.000,E1 267.879} C_DIS
LIN {X 0.146,Y -432.384,Z 859.487,A 0.000,B 0.000,C 90.000,E1 267.650} C_DIS
LIN {X -0.075,Y -423.609,Z 859.486,A 0.000,B 0.000,C 90.000,E1 267.535} C_DIS
LIN {X 0.197,Y -413.064,Z 859.486,A 0.000,B 0.000,C 90.000,E1 267.421} C_DIS
LIN {X 0.066,Y -181.042,Z 859.486,A 0.000,B 0.000,C 90.000,E1 267.421} C_DIS
LIN {X -0.021,Y -180.906,Z 859.474,A 0.000,B 0.000,C 90.000,E1 265.412} C_DIS
LIN {X 0.036,Y -180.707,Z 859.470,A 0.000,B 0.000,C 90.000,E1 264.552} C_DIS
LIN {X -0.045,Y -178.793,Z 859.442,A 0.000,B 0.000,C 90.000,E1 259.511} C_DIS
LIN {X 0.032,Y -175.839,Z 859.413,A 0.000,B 0.000,C 90.000,E1 254.393} C_DIS
LIN {X 0.031,Y -172.029,Z 859.385,A 0.000,B 0.000,C 90.000,E1 249.263} C_DIS
LIN {X 0.008,Y -171.456,Z 859.380,A 0.000,B 0.000,C 90.000,E1 248.411} C_DIS
LIN {X -0.012,Y -167.689,Z 859.356,A 0.000,B 0.000,C 90.000,E1 244.101} C_DIS
LIN {X 0.002,Y -166.370,Z 859.346,A 0.000,B 0.000,C 90.000,E1 242.359} C_DIS
LIN {X -0.006,Y -163.100,Z 859.327,A 0.000,B 0.000,C 90.000,E1 238.869} C_DIS
LIN {X 0.044,Y -161.047,Z 859.312,A 0.000,B 0.000,C 90.000,E1 236.215} C_DIS
LIN {X 0.028,Y -157.783,Z 859.293,A 0.000,B 0.000,C 90.000,E1 232.683} C_DIS
LIN {X -0.029,Y -155.820,Z 859.278,A 0.000,B 0.000,C 90.000,E1 230.033} C_DIS
LIN {X -0.072,Y -152.071,Z 859.253,A 0.000,B 0.000,C 90.000,E1 225.567} C_DIS
LIN {X -0.052,Y -150.321,Z 859.238,A 0.000,B 0.000,C 90.000,E1 222.852} C_DIS
LIN {X -0.031,Y -147.064,Z 859.213,A 0.000,B 0.000,C 90.000,E1 218.302} C_DIS
LIN {X 0.077,Y -145.640,Z 859.198,A 0.000,B 0.000,C 90.000,E1 215.518} C_DIS
LIN {X 0.074,Y -143.022,Z 859.172,A 0.000,B 0.000,C 90.000,E1 210.924} C_DIS
LIN {X 0.006,Y -141.648,Z 859.151,A 0.000,B 0.000,C 90.000,E1 207.257} C_DIS
LIN {X 0.056,Y -139.443,Z 859.115,A 0.000,B 0.000,C 90.000,E1 200.737} C_DIS
LIN {X -0.022,Y -139.175,Z 859.105,A 0.000,B 0.000,C 90.000,E1 198.906} C_DIS
LIN {X 0.006,Y -138.319,Z 859.053,A 0.000,B 0.000,C 90.000,E1 189.557} C_DIS
LIN {X 0.015,Y -139.469,Z 859.006,A 0.000,B 0.000,C 90.000,E1 181.146} C_DIS
LIN {X -0.044,Y -141.038,Z 858.975,A 0.000,B 0.000,C 90.000,E1 175.584} C_DIS
LIN {X 0.051,Y -142.407,Z 858.960,A 0.000,B 0.000,C 90.000,E1 172.761} C_DIS
LIN {X -0.028,Y -144.640,Z 858.934,A 0.000,B 0.000,C 90.000,E1 168.173} C_DIS
LIN {X 0.032,Y -147.836,Z 858.909,A 0.000,B 0.000,C 90.000,E1 163.559} C_DIS
LIN {X -0.025,Y -150.532,Z 858.888,A 0.000,B 0.000,C 90.000,E1 159.934} C_DIS
LIN {X -0.005,Y -153.996,Z 858.868,A 0.000,B 0.000,C 90.000,E1 156.305} C_DIS
LIN {X -0.085,Y -157.409,Z 858.848,A 0.000,B 0.000,C 90.000,E1 152.743} C_DIS
LIN {X -0.005,Y -161.619,Z 858.829,A 0.000,B 0.000,C 90.000,E1 149.154} C_DIS
LIN {X 0.096,Y -165.815,Z 858.809,A 0.000,B 0.000,C 90.000,E1 145.595} C_DIS
LIN {X -0.015,Y -170.782,Z 858.790,A 0.000,B 0.000,C 90.000,E1 142.145} C_DIS
LIN {X 0.007,Y -175.653,Z 858.771,A 0.000,B 0.000,C 90.000,E1 138.690} C_DIS
LIN {X 0.004,Y -181.268,Z 858.752,A 0.000,B 0.000,C 90.000,E1 135.283} C_DIS
LIN {X 0.004,Y -186.742,Z 858.733,A 0.000,B 0.000,C 90.000,E1 131.919} C_DIS
LIN {X -0.044,Y -191.339,Z 858.719,A 0.000,B 0.000,C 90.000,E1 129.439} C_DIS
LIN {X 0.106,Y -193.026,Z 858.713,A 0.000,B 0.000,C 90.000,E1 128.382} C_DIS
LIN {X 0.110,Y -293.597,Z 858.713,A 0.000,B 0.000,C 90.000,E1 128.382} C_DIS
LIN {X 0.061,Y -294.621,Z 858.713,A 0.000,B 0.000,C 90.000,E1 128.382} C_DIS
LIN {X -0.091,Y -298.957,Z 858.712,A 0.000,B 0.000,C 90.000,E1 128.257} C_DIS
LIN {X -0.057,Y -301.177,Z 858.712,A 0.000,B 0.000,C 90.000,E1 128.096} C_DIS
LIN {X -0.178,Y -304.208,Z 858.710,A 0.000,B 0.000,C 90.000,E1 127.810} C_DIS
LIN {X -0.002,Y -307.835,Z 858.707,A 0.000,B 0.000,C 90.000,E1 127.202} C_DIS
LIN {X 0.019,Y -309.281,Z 858.705,A 0.000,B 0.000,C 90.000,E1 126.870} C_DIS
LIN {X 0.042,Y -310.416,Z 858.703,A 0.000,B 0.000,C 90.000,E1 126.537} C_DIS
LIN {X 0.106,Y -320.475,Z 858.685,A 0.000,B 0.000,C 90.000,E1 123.293} C_DIS
LIN {X -0.048,Y -330.835,Z 858.669,A 0.000,B 0.000,C 90.000,E1 120.463} C_DIS
LIN {X 0.043,Y -342.545,Z 858.654,A 0.000,B 0.000,C 90.000,E1 117.641} C_DIS
LIN {X 0.003,Y -355.704,Z 858.638,A 0.000,B 0.000,C 90.000,E1 114.899} C_DIS
LIN {X -0.046,Y -368.715,Z 858.625,A 0.000,B 0.000,C 90.000,E1 112.514} C_DIS
LIN {X -0.058,Y -383.057,Z 858.612,A 0.000,B 0.000,C 90.000,E1 110.174} C_DIS
LIN {X 0.027,Y -398.832,Z 858.599,A 0.000,B 0.000,C 90.000,E1 107.873} C_DIS
LIN {X -0.120,Y -416.155,Z 858.587,A 0.000,B 0.000,C 90.000,E1 105.662} C_DIS
LIN {X -0.048,Y -435.140,Z 858.575,A 0.000,B 0.000,C 90.000,E1 103.480} C_DIS
LIN {X 0.074,Y -455.214,Z 858.564,A 0.000,B 0.000,C 90.000,E1 101.422} C_DIS
LIN {X -0.104,Y -467.944,Z 858.557,A 0.000,B 0.000,C 90.000,E1 100.254} C_DIS
LIN {X -0.134,Y -469.893,Z 858.556,A 0.000,B 0.000,C 90.000,E1 100.018} C_DIS
LIN {X -0.165,Y -471.375,Z 858.554,A 0.000,B 0.000,C 90.000,E1 99.782} C_DIS
LIN {X 0.075,Y -472.561,Z 858.553,A 0.000,B 0.000,C 90.000,E1 99.500} C_DIS
LIN {X -0.071,Y -473.425,Z 858.551,A 0.000,B 0.000,C 90.000,E1 99.265} C_DIS
LIN {X 0.043,Y -474.336,Z 858.549,A 0.000,B 0.000,C 90.000,E1 98.746} C_DIS
LIN {X 0.233,Y -474.271,Z 858.546,A 0.000,B 0.000,C 90.000,E1 98.219} C_DIS
LIN {X -0.110,Y -473.223,Z 858.543,A 0.000,B 0.000,C 90.000,E1 97.757} C_DIS
LIN {X 0.156,Y -472.284,Z 858.542,A 0.000,B 0.000,C 90.000,E1 97.473} C_DIS
LIN {X 0.016,Y -471.012,Z 858.540,A 0.000,B 0.000,C 90.000,E1 97.239} C_DIS
LIN {X -0.055,Y -454.937,Z 858.526,A 0.000,B 0.000,C 90.000,E1 94.702} C_DIS
LIN {X -0.146,Y -442.883,Z 858.515,A 0.000,B 0.000,C 90.000,E1 92.636} C_DIS
LIN {X -0.129,Y -435.137,Z 858.507,A 0.000,B 0.000,C 90.000,E1 91.318} C_DIS
LIN {X -0.092,Y -425.520,Z 858.498,A 0.000,B 0.000,C 90.000,E1 89.714} C_DIS
LIN {X -0.111,Y -414.134,Z 858.488,A 0.000,B 0.000,C 90.000,E1 87.822} C_DIS
LIN {X -0.021,Y -404.325,Z 858.479,A 0.000,B 0.000,C 90.000,E1 86.159} C_DIS
LIN {X -0.029,Y -392.903,Z 858.468,A 0.000,B 0.000,C 90.000,E1 84.204} C_DIS
LIN {X 0.180,Y -380.083,Z 858.455,A 0.000,B 0.000,C 90.000,E1 81.894} C_DIS
LIN {X 0.126,Y -367.414,Z 858.442,A 0.000,B 0.000,C 90.000,E1 79.577} C_DIS
LIN {X 0.025,Y -356.601,Z 858.431,A 0.000,B 0.000,C 90.000,E1 77.521} C_DIS
LIN {X 0.043,Y -345.779,Z 858.419,A 0.000,B 0.000,C 90.000,E1 75.408} C_DIS
LIN {X -0.017,Y -333.496,Z 858.405,A 0.000,B 0.000,C 90.000,E1 72.960} C_DIS
LIN {X 0.095,Y -320.101,Z 858.390,A 0.000,B 0.000,C 90.000,E1 70.115} C_DIS
LIN {X 0.139,Y -308.643,Z 858.375,A 0.000,B 0.000,C 90.000,E1 67.539} C_DIS
LIN {X -0.143,Y -297.440,Z 858.361,A 0.000,B 0.000,C 90.000,E1 64.973} C_DIS
LIN {X -0.045,Y -286.448,Z 858.346,A 0.000,B 0.000,C 90.000,E1 62.281} C_DIS
LIN {X 0.039,Y -275.571,Z 858.331,A 0.000,B 0.000,C 90.000,E1 59.537} C_DIS
LIN {X -0.136,Y -262.608,Z 858.311,A 0.000,B 0.000,C 90.000,E1 56.087} C_DIS
LIN {X 0.033,Y -250.745,Z 858.292,A 0.000,B 0.000,C 90.000,E1 52.477} C_DIS
LIN {X 0.111,Y -241.976,Z 858.275,A 0.000,B 0.000,C 90.000,E1 49.542} C_DIS
LIN {X -0.141,Y -231.914,Z 858.255,A 0.000,B 0.000,C 90.000,E1 45.891} C_DIS
LIN {X -0.045,Y -222.516,Z 858.234,A 0.000,B 0.000,C 90.000,E1 42.081} C_DIS
LIN {X -0.019,Y -215.437,Z 858.217,A 0.000,B 0.000,C 90.000,E1 38.991} C_DIS
LIN {X -0.100,Y -208.778,Z 858.199,A 0.000,B 0.000,C 90.000,E1 35.884} C_DIS
LIN {X 0.032,Y -202.529,Z 858.182,A 0.000,B 0.000,C 90.000,E1 32.673} C_DIS
LIN {X 0.016,Y -196.806,Z 858.164,A 0.000,B 0.000,C 90.000,E1 29.461} C_DIS
LIN {X -0.082,Y -191.756,Z 858.146,A 0.000,B 0.000,C 90.000,E1 26.232} C_DIS
LIN {X 0.052,Y -187.365,Z 858.127,A 0.000,B 0.000,C 90.000,E1 22.898} C_DIS
LIN {X 0.087,Y -183.058,Z 858.104,A 0.000,B 0.000,C 90.000,E1 18.725} C_DIS
LIN {X 0.047,Y -179.905,Z 858.081,A 0.000,B 0.000,C 90.000,E1 14.537} C_DIS
LIN {X 0.002,Y -177.286,Z 858.048,A 0.000,B 0.000,C 90.000,E1 8.624} C_DIS
LIN {X -0.088,Y -178.260,Z 857.979,A 0.000,B 0.000,C 90.000,E1 356.159} C_DIS
LIN {X 0.070,Y -181.085,Z 857.950,A 0.000,B 0.000,C 90.000,E1 351.027} C_DIS
LIN {X 0.057,Y -184.586,Z 857.927,A 0.000,B 0.000,C 90.000,E1 346.825} C_DIS
LIN {X 0.007,Y -189.127,Z 857.904,A 0.000,B 0.000,C 90.000,E1 342.670} C_DIS
LIN {X 0.021,Y -194.659,Z 857.881,A 0.000,B 0.000,C 90.000,E1 338.539} C_DIS
LIN {X 0.038,Y -201.105,Z 857.858,A 0.000,B 0.000,C 90.000,E1 334.460} C_DIS
LIN {X -0.020,Y -208.257,Z 857.836,A 0.000,B 0.000,C 90.000,E1 330.461} C_DIS
LIN {X 0.011,Y -216.135,Z 857.814,A 0.000,B 0.000,C 90.000,E1 326.501} C_DIS
LIN {X -0.104,Y -223.040,Z 857.797,A 0.000,B 0.000,C 90.000,E1 323.417} C_DIS
LIN {X 0.139,Y -231.678,Z 857.777,A 0.000,B 0.000,C 90.000,E1 319.908} C_DIS
LIN {X 0.102,Y -241.199,Z 857.759,A 0.000,B 0.000,C 90.000,E1 316.539} C_DIS
LIN {X -0.023,Y -251.781,Z 857.740,A 0.000,B 0.000,C 90.000,E1 313.257} C_DIS
LIN {X -0.005,Y -263.401,Z 857.722,A 0.000,B 0.000,C 90.000,E1 310.011} C_DIS
LIN {X -0.130,Y -276.005,Z 857.705,A 0.000,B 0.000,C 90.000,E1 306.870} C_DIS
LIN {X -0.172,Y -289.785,Z 857.688,A 0.000,B 0.000,C 90.000,E1 303.785} C_DIS
LIN {X -0.012,Y -306.578,Z 857.669,A 0.000,B 0.000,C 90.000,E1 300.413} C_DIS
LIN {X -0.110,Y -319.556,Z 857.656,A 0.000,B 0.000,C 90.000,E1 298.153} C_DIS
LIN {X 0.048,Y -333.863,Z 857.644,A 0.000,B 0.000,C 90.000,E1 295.899} C_DIS
LIN {X 0.004,Y -355.995,Z 857.627,A 0.000,B 0.000,C 90.000,E1 292.823} C_DIS
LIN {X -0.030,Y -372.912,Z 857.615,A 0.000,B 0.000,C 90.000,E1 290.737} C_DIS
LIN {X 0.078,Y -395.928,Z 857.601,A 0.000,B 0.000,C 90.000,E1 288.181} C_DIS
LIN {X 0.187,Y -413.693,Z 857.591,A 0.000,B 0.000,C 90.000,E1 286.315} C_DIS
LIN {X -0.031,Y -426.260,Z 857.583,A 0.000,B 0.000,C 90.000,E1 285.009} C_DIS
LIN {X -0.062,Y -436.092,Z 857.577,A 0.000,B 0.000,C 90.000,E1 283.939} C_DIS
LIN {X -0.113,Y -445.550,Z 857.571,A 0.000,B 0.000,C 90.000,E1 282.883} C_DIS
LIN {X -0.051,Y -454.381,Z 857.566,A 0.000,B 0.000,C 90.000,E1 281.827} C_DIS
LIN {X 0.029,Y -462.717,Z 857.560,A 0.000,B 0.000,C 90.000,E1 280.782} C_DIS
LIN {X -0.166,Y -470.401,Z 857.554,A 0.000,B 0.000,C 90.000,E1 279.782} C_DIS
LIN {X 0.248,Y -475.680,Z 857.550,A 0.000,B 0.000,C 90.000,E1 278.973} C_DIS
LIN {X 0.238,Y -480.377,Z 857.546,A 0.000,B 0.000,C 90.000,E1 278.219} C_DIS
LIN {X 0.210,Y -484.383,Z 857.542,A 0.000,B 0.000,C 90.000,E1 277.473} C_DIS
LIN {X -0.205,Y -487.614,Z 857.538,A 0.000,B 0.000,C 90.000,E1 276.777} C_DIS
LIN {X -0.001,Y -489.378,Z 857.535,A 0.000,B 0.000,C 90.000,E1 276.258} C_DIS
LIN {X 0.208,Y -490.824,Z 857.532,A 0.000,B 0.000,C 90.000,E1 275.739} C_DIS
LIN {X -0.062,Y -491.906,Z 857.529,A 0.000,B 0.000,C 90.000,E1 275.277} C_DIS
LIN {X 0.165,Y -492.638,Z 857.527,A 0.000,B 0.000,C 90.000,E1 274.759} C_DIS
LIN {X -0.132,Y -492.991,Z 857.524,A 0.000,B 0.000,C 90.000,E1 274.302} C_DIS
LIN {X 0.103,Y -492.896,Z 857.521,A 0.000,B 0.000,C 90.000,E1 273.784} C_DIS
LIN {X -0.183,Y -492.442,Z 857.518,A 0.000,B 0.000,C 90.000,E1 273.326} C_DIS
LIN {X 0.051,Y -491.511,Z 857.516,A 0.000,B 0.000,C 90.000,E1 272.808} C_DIS
LIN {X -0.233,Y -490.164,Z 857.513,A 0.000,B 0.000,C 90.000,E1 272.350} C_DIS
LIN {X -0.030,Y -488.329,Z 857.510,A 0.000,B 0.000,C 90.000,E1 271.835} C_DIS
LIN {X 0.177,Y -485.914,Z 857.507,A 0.000,B 0.000,C 90.000,E1 271.318} C_DIS
LIN {X -0.131,Y -482.913,Z 857.505,A 0.000,B 0.000,C 90.000,E1 270.859} C_DIS
LIN {X 0.031,Y -479.255,Z 857.502,A 0.000,B 0.000,C 90.000,E1 270.344} C_DIS
LIN {X 0.171,Y -474.766,Z 857.499,A 0.000,B 0.000,C 90.000,E1 269.828} C_DIS
LIN {X -0.183,Y -469.387,Z 857.496,A 0.000,B 0.000,C 90.000,E1 269.370} C_DIS
LIN {X -0.188,Y -463.368,Z 857.494,A 0.000,B 0.000,C 90.000,E1 268.912} C_DIS
LIN {X -0.177,Y -456.720,Z 857.492,A 0.000,B 0.000,C 90.000,E1 268.511} C_DIS
LIN {X -0.051,Y -449.659,Z 857.490,A 0.000,B 0.000,C 90.000,E1 268.165} C_DIS
LIN {X 0.133,Y -442.236,Z 857.488,A 0.000,B 0.000,C 90.000,E1 267.879} C_DIS
LIN {X -0.125,Y -434.486,Z 857.487,A 0.000,B 0.000,C 90.000,E1 267.707} C_DIS
LIN {X 0.023,Y -426.271,Z 857.486,A 0.000,B 0.000,C 90.000,E1 267.535} C_DIS
LIN {X -0.165,Y -418.737,Z 857.486,A 0.000,B 0.000,C 90.000,E1 267.478} C_DIS
LIN {X 0.050,Y -412.792,Z 857.486,A 0.000,B 0.000,C 90.000,E1 267.421} C_DIS
LIN {X 0.001,Y -181.040,Z 857.486,A 0.000,B 0.000,C 90.000,E1 267.421} C_DIS
LIN {X 0.024,Y -180.820,Z 857.471,A 0.000,B 0.000,C 90.000,E1 264.837} C_DIS
LIN {X -0.075,Y -178.923,Z 857.443,A 0.000,B 0.000,C 90.000,E1 259.803} C_DIS
LIN {X -0.037,Y -175.969,Z 857.415,A 0.000,B 0.000,C 90.000,E1 254.700} C_DIS
LIN {X -0.043,Y -175.452,Z 857.410,A 0.000,B 0.000,C 90.000,E1 253.850} C_DIS
LIN {X -0.034,Y -172.205,Z 857.386,A 0.000,B 0.000,C 90.000,E1 249.571} C_DIS
LIN {X -0.057,Y -171.679,Z 857.382,A 0.000,B 0.000,C 90.000,E1 248.720} C_DIS
LIN {X -0.066,Y -167.905,Z 857.358,A 0.000,B 0.000,C 90.000,E1 244.409} C_DIS
LIN {X -0.047,Y -166.647,Z 857.348,A 0.000,B 0.000,C 90.000,E1 242.666} C_DIS
LIN {X 0.008,Y -162.630,Z 857.324,A 0.000,B 0.000,C 90.000,E1 238.280} C_DIS
LIN {X 0.067,Y -161.317,Z 857.314,A 0.000,B 0.000,C 90.000,E1 236.501} C_DIS
LIN {X -0.024,Y -157.314,Z 857.289,A 0.000,B 0.000,C 90.000,E1 232.110} C_DIS
LIN {X -0.090,Y -155.293,Z 857.275,A 0.000,B 0.000,C 90.000,E1 229.461} C_DIS
LIN {X 0.056,Y -151.655,Z 857.250,A 0.000,B 0.000,C 90.000,E1 224.919} C_DIS
LIN {X -0.007,Y -150.522,Z 857.240,A 0.000,B 0.000,C 90.000,E1 223.137} C_DIS
LIN {X 0.016,Y -147.246,Z 857.214,A 0.000,B 0.000,C 90.000,E1 218.588} C_DIS
LIN {X -0.019,Y -145.271,Z 857.194,A 0.000,B 0.000,C 90.000,E1 214.945} C_DIS
LIN {X 0.016,Y -142.378,Z 857.163,A 0.000,B 0.000,C 90.000,E1 209.411} C_DIS
LIN {X 0.064,Y -141.354,Z 857.148,A 0.000,B 0.000,C 90.000,E1 206.616} C_DIS
LIN {X 0.047,Y -139.341,Z 857.112,A 0.000,B 0.000,C 90.000,E1 200.120} C_DIS
LIN {X -0.034,Y -139.008,Z 857.102,A 0.000,B 0.000,C 90.000,E1 198.290} C_DIS
LIN {X 0.054,Y -138.340,Z 857.055,A 0.000,B 0.000,C 90.000,E1 189.849} C_DIS
LIN {X -0.063,Y -139.402,Z 857.008,A 0.000,B 0.000,C 90.000,E1 181.489} C_DIS
LIN {X -0.009,Y -141.308,Z 856.972,A 0.000,B 0.000,C 90.000,E1 174.951} C_DIS
LIN {X -0.052,Y -142.669,Z 856.956,A 0.000,B 0.000,C 90.000,E1 172.186} C_DIS
LIN {X 0.070,Y -145.018,Z 856.931,A 0.000,B 0.000,C 90.000,E1 167.521} C_DIS
LIN {X 0.027,Y -147.645,Z 856.910,A 0.000,B 0.000,C 90.000,E1 163.866} C_DIS
LIN {X -0.037,Y -150.279,Z 856.890,A 0.000,B 0.000,C 90.000,E1 160.242} C_DIS
LIN {X -0.024,Y -153.682,Z 856.870,A 0.000,B 0.000,C 90.000,E1 156.613} C_DIS
LIN {X 0.031,Y -157.096,Z 856.850,A 0.000,B 0.000,C 90.000,E1 152.999} C_DIS
LIN {X -0.031,Y -161.235,Z 856.830,A 0.000,B 0.000,C 90.000,E1 149.459} C_DIS
LIN {X 0.055,Y -163.322,Z 856.820,A 0.000,B 0.000,C 90.000,E1 147.661} C_DIS
LIN {X -0.074,Y -167.774,Z 856.801,A 0.000,B 0.000,C 90.000,E1 144.196} C_DIS
LIN {X 0.077,Y -171.589,Z 856.786,A 0.000,B 0.000,C 90.000,E1 141.537} C_DIS
LIN {X 0.008,Y -176.541,Z 856.767,A 0.000,B 0.000,C 90.000,E1 138.119} C_DIS
LIN {X 0.001,Y -180.839,Z 856.753,A 0.000,B 0.000,C 90.000,E1 135.567} C_DIS
LIN {X -0.015,Y -186.249,Z 856.734,A 0.000,B 0.000,C 90.000,E1 132.204} C_DIS
LIN {X -0.077,Y -190.886,Z 856.721,A 0.000,B 0.000,C 90.000,E1 129.725} C_DIS
LIN {X 0.010,Y -193.013,Z 856.713,A 0.000,B 0.000,C 90.000,E1 128.418} C_DIS
LIN {X 0.168,Y -293.811,Z 856.713,A 0.000,B 0.000,C 90.000,E1 128.382} C_DIS
LIN {X -0.042,Y -296.077,Z 856.713,A 0.000,B 0.000,C 90.000,E1 128.382} C_DIS
LIN {X -0.002,Y -301.675,Z 856.711,A 0.000,B 0.000,C 90.000,E1 128.051} C_DIS
LIN {X 0.067,Y -304.866,Z 856.709,A 0.000,B 0.000,C 90.000,E1 127.684} C_DIS
LIN {X 0.149,Y -306.844,Z 856.708,A 0.000,B 0.000,C 90.000,E1 127.363} C_DIS
LIN {X 0.044,Y -308.393,Z 856.706,A 0.000,B 0.000,C 90.000,E1 127.076} C_DIS
LIN {X 0.074,Y -309.702,Z 856.704,A 0.000,B 0.000,C 90.000,E1 126.744} C_DIS
LIN {X 0.000,Y -321.926,Z 856.683,A 0.000,B 0.000,C 90.000,E1 122.880} C_DIS
LIN {X 0.165,Y -332.484,Z 856.667,A 0.000,B 0.000,C 90.000,E1 120.001} C_DIS
LIN {X -0.149,Y -344.402,Z 856.651,A 0.000,B 0.000,C 90.000,E1 117.257} C_DIS
LIN {X -0.148,Y -357.792,Z 856.636,A 0.000,B 0.000,C 90.000,E1 114.515} C_DIS
LIN {X 0.050,Y -371.021,Z 856.623,A 0.000,B 0.000,C 90.000,E1 112.099} C_DIS
LIN {X 0.110,Y -385.597,Z 856.610,A 0.000,B 0.000,C 90.000,E1 109.758} C_DIS
LIN {X -0.110,Y -401.627,Z 856.597,A 0.000,B 0.000,C 90.000,E1 107.511} C_DIS
LIN {X 0.207,Y -419.224,Z 856.585,A 0.000,B 0.000,C 90.000,E1 105.245} C_DIS
LIN {X -0.036,Y -438.479,Z 856.573,A 0.000,B 0.000,C 90.000,E1 103.119} C_DIS
LIN {X -0.225,Y -458.652,Z 856.562,A 0.000,B 0.000,C 90.000,E1 101.130} C_DIS
LIN {X 0.210,Y -466.345,Z 856.558,A 0.000,B 0.000,C 90.000,E1 100.366} C_DIS
LIN {X 0.148,Y -468.658,Z 856.556,A 0.000,B 0.000,C 90.000,E1 100.141} C_DIS
LIN {X 0.038,Y -470.503,Z 856.555,A 0.000,B 0.000,C 90.000,E1 99.905} C_DIS
LIN {X -0.073,Y -471.895,Z 856.554,A 0.000,B 0.000,C 90.000,E1 99.670} C_DIS
LIN {X 0.027,Y -473.704,Z 856.551,A 0.000,B 0.000,C 90.000,E1 99.151} C_DIS
LIN {X 0.210,Y -474.423,Z 856.548,A 0.000,B 0.000,C 90.000,E1 98.624} C_DIS
LIN {X -0.138,Y -474.173,Z 856.545,A 0.000,B 0.000,C 90.000,E1 98.163} C_DIS
LIN {X -0.011,Y -472.923,Z 856.542,A 0.000,B 0.000,C 90.000,E1 97.644} C_DIS
LIN {X -0.151,Y -471.862,Z 856.541,A 0.000,B 0.000,C 90.000,E1 97.409} C_DIS
LIN {X 0.116,Y -470.442,Z 856.540,A 0.000,B 0.000,C 90.000,E1 97.125} C_DIS
LIN {X -0.235,Y -455.884,Z 856.527,A 0.000,B 0.000,C 90.000,E1 94.878} C_DIS
LIN {X 0.178,Y -443.798,Z 856.515,A 0.000,B 0.000,C 90.000,E1 92.751} C_DIS
LIN {X 0.207,Y -436.101,Z 856.508,A 0.000,B 0.000,C 90.000,E1 91.432} C_DIS
LIN {X -0.175,Y -426.513,Z 856.499,A 0.000,B 0.000,C 90.000,E1 89.885} C_DIS
LIN {X -0.175,Y -415.145,Z 856.489,A 0.000,B 0.000,C 90.000,E1 87.993} C_DIS
LIN {X 0.001,Y -403.686,Z 856.478,A 0.000,B 0.000,C 90.000,E1 86.045} C_DIS
LIN {X -0.023,Y -392.258,Z 856.467,A 0.000,B 0.000,C 90.000,E1 84.090} C_DIS
LIN {X 0.167,Y -379.449,Z 856.454,A 0.000,B 0.000,C 90.000,E1 81.781} C_DIS
LIN {X 0.161,Y -366.804,Z 856.442,A 0.000,B 0.000,C 90.000,E1 79.454} C_DIS
LIN {X -0.024,Y -356.017,Z 856.430,A 0.000,B 0.000,C 90.000,E1 77.409} C_DIS
LIN {X 0.055,Y -346.762,Z 856.420,A 0.000,B 0.000,C 90.000,E1 75.589} C_DIS
LIN {X 0.026,Y -336.029,Z 856.408,A 0.000,B 0.000,C 90.000,E1 73.449} C_DIS
LIN {X -0.066,Y -324.013,Z 856.394,A 0.000,B 0.000,C 90.000,E1 70.967} C_DIS
LIN {X -0.033,Y -312.452,Z 856.380,A 0.000,B 0.000,C 90.000,E1 68.411} C_DIS
LIN {X 0.055,Y -301.167,Z 856.366,A 0.000,B 0.000,C 90.000,E1 65.793} C_DIS
LIN {X -0.142,Y -291.528,Z 856.353,A 0.000,B 0.000,C 90.000,E1 63.512} C_DIS
LIN {X 0.001,Y -283.367,Z 856.341,A 0.000,B 0.000,C 90.000,E1 61.463} C_DIS
LIN {X -0.101,Y -272.633,Z 856.326,A 0.000,B 0.000,C 90.000,E1 58.742} C_DIS
LIN {X 0.146,Y -259.976,Z 856.307,A 0.000,B 0.000,C 90.000,E1 55.182} C_DIS
LIN {X 0.023,Y -248.393,Z 856.287,A 0.000,B 0.000,C 90.000,E1 51.618} C_DIS
LIN {X -0.010,Y -237.826,Z 856.266,A 0.000,B 0.000,C 90.000,E1 47.957} C_DIS
LIN {X 0.093,Y -228.063,Z 856.246,A 0.000,B 0.000,C 90.000,E1 44.190} C_DIS
LIN {X 0.069,Y -218.971,Z 856.224,A 0.000,B 0.000,C 90.000,E1 40.378} C_DIS
LIN {X 0.009,Y -210.425,Z 856.203,A 0.000,B 0.000,C 90.000,E1 36.503} C_DIS
LIN {X -0.002,Y -202.580,Z 856.181,A 0.000,B 0.000,C 90.000,E1 32.546} C_DIS
LIN {X -0.015,Y -196.865,Z 856.163,A 0.000,B 0.000,C 90.000,E1 29.333} C_DIS
LIN {X 0.063,Y -191.842,Z 856.145,A 0.000,B 0.000,C 90.000,E1 26.052} C_DIS
LIN {X 0.027,Y -187.492,Z 856.127,A 0.000,B 0.000,C 90.000,E1 22.770} C_DIS
LIN {X 0.063,Y -183.220,Z 856.103,A 0.000,B 0.000,C 90.000,E1 18.598} C_DIS
LIN {X 0.024,Y -180.103,Z 856.080,A 0.000,B 0.000,C 90.000,E1 14.411} C_DIS
LIN {X -0.048,Y -177.579,Z 856.047,A 0.000,B 0.000,C 90.000,E1 8.511} C_DIS
LIN {X -0.079,Y -178.580,Z 855.979,A 0.000,B 0.000,C 90.000,E1 356.159} C_DIS
LIN {X -0.088,Y -181.426,Z 855.950,A 0.000,B 0.000,C 90.000,E1 351.084} C_DIS
LIN {X -0.091,Y -184.942,Z 855.927,A 0.000,B 0.000,C 90.000,E1 346.881} C_DIS
LIN {X 0.050,Y -189.488,Z 855.904,A 0.000,B 0.000,C 90.000,E1 342.670} C_DIS
LIN {X 0.077,Y -194.976,Z 855.881,A 0.000,B 0.000,C 90.000,E1 338.539} C_DIS
LIN {X 0.019,Y -201.387,Z 855.858,A 0.000,B 0.000,C 90.000,E1 334.485} C_DIS
LIN {X 0.058,Y -208.543,Z 855.836,A 0.000,B 0.000,C 90.000,E1 330.461} C_DIS
LIN {X 0.101,Y -216.384,Z 855.814,A 0.000,B 0.000,C 90.000,E1 326.501} C_DIS
LIN {X -0.004,Y -223.275,Z 855.797,A 0.000,B 0.000,C 90.000,E1 323.417} C_DIS
LIN {X -0.076,Y -231.915,Z 855.778,A 0.000,B 0.000,C 90.000,E1 319.989} C_DIS
LIN {X 0.049,Y -241.414,Z 855.759,A 0.000,B 0.000,C 90.000,E1 316.581} C_DIS
LIN {X -0.073,Y -251.934,Z 855.740,A 0.000,B 0.000,C 90.000,E1 313.299} C_DIS
LIN {X 0.140,Y -263.534,Z 855.722,A 0.000,B 0.000,C 90.000,E1 310.011} C_DIS
LIN {X 0.025,Y -276.092,Z 855.705,A 0.000,B 0.000,C 90.000,E1 306.870} C_DIS
LIN {X -0.007,Y -289.837,Z 855.688,A 0.000,B 0.000,C 90.000,E1 303.785} C_DIS
LIN {X -0.102,Y -306.538,Z 855.669,A 0.000,B 0.000,C 90.000,E1 300.463} C_DIS
LIN {X 0.071,Y -319.458,Z 855.656,A 0.000,B 0.000,C 90.000,E1 298.153} C_DIS
LIN {X 0.132,Y -331.549,Z 855.646,A 0.000,B 0.000,C 90.000,E1 296.232} C_DIS
LIN {X 0.029,Y -353.410,Z 855.629,A 0.000,B 0.000,C 90.000,E1 293.153} C_DIS
LIN {X -0.151,Y -372.474,Z 855.615,A 0.000,B 0.000,C 90.000,E1 290.791} C_DIS
LIN {X 0.129,Y -395.700,Z 855.601,A 0.000,B 0.000,C 90.000,E1 288.181} C_DIS
LIN {X 0.124,Y -413.562,Z 855.591,A 0.000,B 0.000,C 90.000,E1 286.315} C_DIS
LIN {X -0.082,Y -426.130,Z 855.583,A 0.000,B 0.000,C 90.000,E1 285.009} C_DIS
LIN {X -0.111,Y -435.976,Z 855.577,A 0.000,B 0.000,C 90.000,E1 283.939} C_DIS
LIN {X -0.165,Y -445.446,Z 855.571,A 0.000,B 0.000,C 90.000,E1 282.883} C_DIS
LIN {X -0.105,Y -454.282,Z 855.566,A 0.000,B 0.000,C 90.000,E1 281.827} C_DIS
LIN {X -0.027,Y -462.619,Z 855.560,A 0.000,B 0.000,C 90.000,E1 280.782} C_DIS
LIN {X 0.239,Y -470.339,Z 855.554,A 0.000,B 0.000,C 90.000,E1 279.726} C_DIS
LIN {X 0.188,Y -475.621,Z 855.550,A 0.000,B 0.000,C 90.000,E1 278.973} C_DIS
LIN {X 0.178,Y -480.327,Z 855.546,A 0.000,B 0.000,C 90.000,E1 278.219} C_DIS
LIN {X 0.149,Y -484.346,Z 855.542,A 0.000,B 0.000,C 90.000,E1 277.473} C_DIS
LIN {X 0.218,Y -487.567,Z 855.537,A 0.000,B 0.000,C 90.000,E1 276.720} C_DIS
LIN {X -0.065,Y -489.330,Z 855.535,A 0.000,B 0.000,C 90.000,E1 276.258} C_DIS
LIN {X 0.145,Y -490.787,Z 855.532,A 0.000,B 0.000,C 90.000,E1 275.739} C_DIS
LIN {X -0.125,Y -491.875,Z 855.529,A 0.000,B 0.000,C 90.000,E1 275.277} C_DIS
LIN {X 0.102,Y -492.605,Z 855.526,A 0.000,B 0.000,C 90.000,E1 274.759} C_DIS
LIN {X -0.197,Y -492.938,Z 855.524,A 0.000,B 0.000,C 90.000,E1 274.302} C_DIS
LIN {X 0.039,Y -492.875,Z 855.521,A 0.000,B 0.000,C 90.000,E1 273.784} C_DIS
LIN {X -0.248,Y -492.434,Z 855.518,A 0.000,B 0.000,C 90.000,E1 273.326} C_DIS
LIN {X -0.013,Y -491.533,Z 855.516,A 0.000,B 0.000,C 90.000,E1 272.808} C_DIS
LIN {X 0.192,Y -490.203,Z 855.513,A 0.000,B 0.000,C 90.000,E1 272.293} C_DIS
LIN {X -0.094,Y -488.377,Z 855.510,A 0.000,B 0.000,C 90.000,E1 271.835} C_DIS
LIN {X 0.114,Y -485.961,Z 855.507,A 0.000,B 0.000,C 90.000,E1 271.318} C_DIS
LIN {X -0.193,Y -483.009,Z 855.505,A 0.000,B 0.000,C 90.000,E1 270.859} C_DIS
LIN {X -0.030,Y -479.387,Z 855.502,A 0.000,B 0.000,C 90.000,E1 270.344} C_DIS
LIN {X 0.112,Y -474.953,Z 855.499,A 0.000,B 0.000,C 90.000,E1 269.828} C_DIS
LIN {X 0.228,Y -469.621,Z 855.496,A 0.000,B 0.000,C 90.000,E1 269.312} C_DIS
LIN {X 0.205,Y -463.670,Z 855.494,A 0.000,B 0.000,C 90.000,E1 268.854} C_DIS
LIN {X 0.156,Y -457.001,Z 855.492,A 0.000,B 0.000,C 90.000,E1 268.453} C_DIS
LIN {X 0.230,Y -449.781,Z 855.490,A 0.000,B 0.000,C 90.000,E1 268.108} C_DIS
LIN {X -0.044,Y -442.458,Z 855.488,A 0.000,B 0.000,C 90.000,E1 267.879} C_DIS
LIN {X 0.112,Y -434.488,Z 855.487,A 0.000,B 0.000,C 90.000,E1 267.650} C_DIS
LIN {X -0.178,Y -425.746,Z 855.486,A 0.000,B 0.000,C 90.000,E1 267.535} C_DIS
LIN {X 0.088,Y -418.488,Z 855.486,A 0.000,B 0.000,C 90.000,E1 267.421} C_DIS
LIN {X -0.102,Y -412.300,Z 855.486,A 0.000,B 0.000,C 90.000,E1 267.421} C_DIS
LIN {X -0.065,Y -181.037,Z 855.486,A 0.000,B 0.000,C 90.000,E1 267.421} C_DIS
LIN {X -0.038,Y -180.813,Z 855.471,A 0.000,B 0.000,C 90.000,E1 264.837} C_DIS
LIN {X 0.040,Y -178.915,Z 855.443,A 0.000,B 0.000,C 90.000,E1 259.746} C_DIS
LIN {X -0.051,Y -175.960,Z 855.415,A 0.000,B 0.000,C 90.000,E1 254.685} C_DIS
LIN {X 0.065,Y -175.434,Z 855.410,A 0.000,B 0.000,C 90.000,E1 253.795} C_DIS
LIN {X 0.067,Y -172.192,Z 855.386,A 0.000,B 0.000,C 90.000,E1 249.518} C_DIS
LIN {X 0.044,Y -171.666,Z 855.382,A 0.000,B 0.000,C 90.000,E1 248.666} C_DIS
LIN {X 0.027,Y -167.890,Z 855.358,A 0.000,B 0.000,C 90.000,E1 244.357} C_DIS
LIN {X 0.042,Y -166.629,Z 855.348,A 0.000,B 0.000,C 90.000,E1 242.615} C_DIS
LIN {X 0.036,Y -162.614,Z 855.324,A 0.000,B 0.000,C 90.000,E1 238.250} C_DIS
LIN {X 0.010,Y -161.300,Z 855.314,A 0.000,B 0.000,C 90.000,E1 236.501} C_DIS
LIN {X 0.044,Y -157.298,Z 855.289,A 0.000,B 0.000,C 90.000,E1 232.065} C_DIS
LIN {X 0.072,Y -155.273,Z 855.274,A 0.000,B 0.000,C 90.000,E1 229.380} C_DIS
LIN {X 0.000,Y -151.640,Z 855.250,A 0.000,B 0.000,C 90.000,E1 224.919} C_DIS
LIN {X 0.047,Y -150.509,Z 855.240,A 0.000,B 0.000,C 90.000,E1 223.095} C_DIS
LIN {X -0.038,Y -147.234,Z 855.214,A 0.000,B 0.000,C 90.000,E1 218.588} C_DIS
LIN {X 0.046,Y -145.257,Z 855.194,A 0.000,B 0.000,C 90.000,E1 214.898} C_DIS
LIN {X -0.038,Y -142.370,Z 855.163,A 0.000,B 0.000,C 90.000,E1 209.411} C_DIS
LIN {X 0.083,Y -141.755,Z 855.153,A 0.000,B 0.000,C 90.000,E1 207.513} C_DIS
LIN {X 0.009,Y -139.496,Z 855.117,A 0.000,B 0.000,C 90.000,E1 201.046} C_DIS
LIN {X 0.045,Y -139.002,Z 855.101,A 0.000,B 0.000,C 90.000,E1 198.236} C_DIS
LIN {X 0.002,Y -138.338,Z 855.055,A 0.000,B 0.000,C 90.000,E1 189.849} C_DIS
LIN {X 0.024,Y -139.408,Z 855.008,A 0.000,B 0.000,C 90.000,E1 181.432} C_DIS
LIN {X -0.063,Y -141.318,Z 854.972,A 0.000,B 0.000,C 90.000,E1 174.951} C_DIS
LIN {X 0.036,Y -142.677,Z 854.956,A 0.000,B 0.000,C 90.000,E1 172.129} C_DIS
LIN {X 0.015,Y -145.032,Z 854.931,A 0.000,B 0.000,C 90.000,E1 167.521} C_DIS
LIN {X -0.028,Y -147.657,Z 854.910,A 0.000,B 0.000,C 90.000,E1 163.866} C_DIS
LIN {X 0.049,Y -150.295,Z 854.890,A 0.000,B 0.000,C 90.000,E1 160.188} C_DIS
LIN {X -0.080,Y -153.704,Z 854.870,A 0.000,B 0.000,C 90.000,E1 156.613} C_DIS
LIN {X -0.026,Y -157.118,Z 854.850,A 0.000,B 0.000,C 90.000,E1 152.999} C_DIS
LIN {X 0.050,Y -161.261,Z 854.830,A 0.000,B 0.000,C 90.000,E1 149.410} C_DIS
LIN {X -0.022,Y -164.380,Z 854.815,A 0.000,B 0.000,C 90.000,E1 146.786} C_DIS
LIN {X -0.035,Y -169.055,Z 854.796,A 0.000,B 0.000,C 90.000,E1 143.290} C_DIS
LIN {X 0.017,Y -171.616,Z 854.786,A 0.000,B 0.000,C 90.000,E1 141.537} C_DIS
LIN {X 0.065,Y -176.572,Z 854.767,A 0.000,B 0.000,C 90.000,E1 138.081} C_DIS
LIN {X -0.061,Y -180.871,Z 854.753,A 0.000,B 0.000,C 90.000,E1 135.567} C_DIS
LIN {X 0.060,Y -186.284,Z 854.734,A 0.000,B 0.000,C 90.000,E1 132.162} C_DIS
LIN {X -0.019,Y -190.919,Z 854.720,A 0.000,B 0.000,C 90.000,E1 129.688} C_DIS
LIN {X -0.114,Y -192.999,Z 854.714,A 0.000,B 0.000,C 90.000,E1 128.463} C_DIS
LIN {X 0.023,Y -293.749,Z 854.713,A 0.000,B 0.000,C 90.000,E1 128.418} C_DIS
LIN {X 0.103,Y -295.192,Z 854.713,A 0.000,B 0.000,C 90.000,E1 128.382} C_DIS
LIN {X -0.024,Y -299.563,Z 854.712,A 0.000,B 0.000,C 90.000,E1 128.222} C_DIS
LIN {X 0.084,Y -301.927,Z 854.711,A 0.000,B 0.000,C 90.000,E1 128.016} C_DIS
LIN {X -0.006,Y -305.774,Z 854.709,A 0.000,B 0.000,C 90.000,E1 127.569} C_DIS
LIN {X 0.030,Y -307.637,Z 854.707,A 0.000,B 0.000,C 90.000,E1 127.237} C_DIS
LIN {X 0.008,Y -309.092,Z 854.705,A 0.000,B 0.000,C 90.000,E1 126.916} C_DIS
LIN {X -0.177,Y -311.191,Z 854.701,A 0.000,B 0.000,C 90.000,E1 126.297} C_DIS
LIN {X -0.014,Y -321.370,Z 854.684,A 0.000,B 0.000,C 90.000,E1 123.038} C_DIS
LIN {X -0.139,Y -331.854,Z 854.668,A 0.000,B 0.000,C 90.000,E1 120.207} C_DIS
LIN {X -0.017,Y -343.699,Z 854.652,A 0.000,B 0.000,C 90.000,E1 117.385} C_DIS
LIN {X -0.026,Y -357.002,Z 854.637,A 0.000,B 0.000,C 90.000,E1 114.643} C_DIS
LIN {X -0.047,Y -370.150,Z 854.624,A 0.000,B 0.000,C 90.000,E1 112.259} C_DIS
LIN {X -0.160,Y -384.641,Z 854.611,A 0.000,B 0.000,C 90.000,E1 109.939} C_DIS
LIN {X -0.033,Y -400.579,Z 854.598,A 0.000,B 0.000,C 90.000,E1 107.638} C_DIS
LIN {X -0.136,Y -418.076,Z 854.586,A 0.000,B 0.000,C 90.000,E1 105.426} C_DIS
LIN {X -0.002,Y -437.233,Z 854.574,A 0.000,B 0.000,C 90.000,E1 103.244} C_DIS
LIN {X -0.178,Y -457.371,Z 854.562,A 0.000,B 0.000,C 90.000,E1 101.243} C_DIS
LIN {X 0.152,Y -467.596,Z 854.557,A 0.000,B 0.000,C 90.000,E1 100.254} C_DIS
LIN {X 0.183,Y -469.590,Z 854.556,A 0.000,B 0.000,C 90.000,E1 100.018} C_DIS
LIN {X -0.048,Y -471.238,Z 854.554,A 0.000,B 0.000,C 90.000,E1 99.792} C_DIS
LIN {X -0.200,Y -472.476,Z 854.553,A 0.000,B 0.000,C 90.000,E1 99.557} C_DIS
LIN {X -0.020,Y -473.995,Z 854.550,A 0.000,B 0.000,C 90.000,E1 99.029} C_DIS
LIN {X 0.093,Y -474.474,Z 854.547,A 0.000,B 0.000,C 90.000,E1 98.511} C_DIS
LIN {X 0.217,Y -473.989,Z 854.545,A 0.000,B 0.000,C 90.000,E1 97.992} C_DIS
LIN {X -0.123,Y -472.471,Z 854.542,A 0.000,B 0.000,C 90.000,E1 97.530} C_DIS
LIN {X 0.204,Y -471.245,Z 854.540,A 0.000,B 0.000,C 90.000,E1 97.239} C_DIS
LIN {X -0.096,Y -453.612,Z 854.525,A 0.000,B 0.000,C 90.000,E1 94.473} C_DIS
LIN {X 0.043,Y -443.071,Z 854.515,A 0.000,B 0.000,C 90.000,E1 92.636} C_DIS
LIN {X 0.063,Y -435.325,Z 854.507,A 0.000,B 0.000,C 90.000,E1 91.318} C_DIS
LIN {X 0.099,Y -425.735,Z 854.498,A 0.000,B 0.000,C 90.000,E1 89.714} C_DIS
LIN {X 0.075,Y -414.341,Z 854.488,A 0.000,B 0.000,C 90.000,E1 87.822} C_DIS
LIN {X 0.164,Y -404.541,Z 854.479,A 0.000,B 0.000,C 90.000,E1 86.159} C_DIS
LIN {X 0.158,Y -393.091,Z 854.468,A 0.000,B 0.000,C 90.000,E1 84.204} C_DIS
LIN {X -0.009,Y -380.248,Z 854.455,A 0.000,B 0.000,C 90.000,E1 81.951} C_DIS
LIN {X -0.051,Y -367.594,Z 854.442,A 0.000,B 0.000,C 90.000,E1 79.634} C_DIS
LIN {X 0.162,Y -355.291,Z 854.429,A 0.000,B 0.000,C 90.000,E1 77.229} C_DIS
LIN {X -0.110,Y -346.045,Z 854.419,A 0.000,B 0.000,C 90.000,E1 75.463} C_DIS
LIN {X 0.166,Y -333.831,Z 854.406,A 0.000,B 0.000,C 90.000,E1 72.960} C_DIS
LIN {X -0.135,Y -320.477,Z 854.390,A 0.000,B 0.000,C 90.000,E1 70.188} C_DIS
LIN {X -0.081,Y -309.011,Z 854.376,A 0.000,B 0.000,C 90.000,E1 67.614} C_DIS
LIN {X 0.042,Y -297.861,Z 854.361,A 0.000,B 0.000,C 90.000,E1 64.973} C_DIS
LIN {X 0.145,Y -286.975,Z 854.346,A 0.000,B 0.000,C 90.000,E1 62.281} C_DIS
LIN {X -0.004,Y -276.191,Z 854.331,A 0.000,B 0.000,C 90.000,E1 59.587} C_DIS
LIN {X 0.072,Y -263.371,Z 854.312,A 0.000,B 0.000,C 90.000,E1 56.087} C_DIS
LIN {X -0.098,Y -251.571,Z 854.292,A 0.000,B 0.000,C 90.000,E1 52.557} C_DIS
LIN {X 0.000,Y -241.768,Z 854.274,A 0.000,B 0.000,C 90.000,E1 49.256} C_DIS
LIN {X -0.097,Y -231.767,Z 854.253,A 0.000,B 0.000,C 90.000,E1 45.567} C_DIS
LIN {X -0.009,Y -222.453,Z 854.232,A 0.000,B 0.000,C 90.000,E1 41.757} C_DIS
LIN {X 0.010,Y -215.423,Z 854.215,A 0.000,B 0.000,C 90.000,E1 38.669} C_DIS
LIN {X 0.050,Y -207.174,Z 854.193,A 0.000,B 0.000,C 90.000,E1 34.739} C_DIS
LIN {X -0.088,Y -201.074,Z 854.175,A 0.000,B 0.000,C 90.000,E1 31.592} C_DIS
LIN {X -0.066,Y -195.551,Z 854.157,A 0.000,B 0.000,C 90.000,E1 28.359} C_DIS
LIN {X -0.020,Y -190.718,Z 854.139,A 0.000,B 0.000,C 90.000,E1 25.079} C_DIS
LIN {X 0.008,Y -186.622,Z 854.121,A 0.000,B 0.000,C 90.000,E1 21.770} C_DIS
LIN {X 0.067,Y -182.651,Z 854.098,A 0.000,B 0.000,C 90.000,E1 17.583} C_DIS
LIN {X 0.066,Y -179.375,Z 854.070,A 0.000,B 0.000,C 90.000,E1 12.535} C_DIS
LIN {X -0.025,Y -177.323,Z 854.027,A 0.000,B 0.000,C 90.000,E1 4.935} C_DIS
LIN {X -0.072,Y -178.901,Z 853.979,A 0.000,B 0.000,C 90.000,E1 356.159} C_DIS
LIN {X -0.068,Y -181.769,Z 853.950,A 0.000,B 0.000,C 90.000,E1 351.084} C_DIS
LIN {X -0.060,Y -185.282,Z 853.927,A 0.000,B 0.000,C 90.000,E1 346.881} C_DIS
LIN {X -0.088,Y -189.820,Z 853.904,A 0.000,B 0.000,C 90.000,E1 342.725} C_DIS
LIN {X -0.050,Y -195.290,Z 853.881,A 0.000,B 0.000,C 90.000,E1 338.592} C_DIS
LIN {X -0.097,Y -201.662,Z 853.858,A 0.000,B 0.000,C 90.000,E1 334.537} C_DIS
LIN {X -0.046,Y -208.806,Z 853.836,A 0.000,B 0.000,C 90.000,E1 330.511} C_DIS
LIN {X 0.009,Y -216.630,Z 853.814,A 0.000,B 0.000,C 90.000,E1 326.548} C_DIS
LIN {X 0.094,Y -223.506,Z 853.797,A 0.000,B 0.000,C 90.000,E1 323.417} C_DIS
LIN {X 0.030,Y -232.128,Z 853.778,A 0.000,B 0.000,C 90.000,E1 319.989} C_DIS
LIN {X -0.004,Y -241.619,Z 853.759,A 0.000,B 0.000,C 90.000,E1 316.620} C_DIS
LIN {X 0.052,Y -252.104,Z 853.741,A 0.000,B 0.000,C 90.000,E1 313.299} C_DIS
LIN {X -0.097,Y -263.663,Z 853.723,A 0.000,B 0.000,C 90.000,E1 310.092} C_DIS
LIN {X 0.169,Y -276.188,Z 853.705,A 0.000,B 0.000,C 90.000,E1 306.870} C_DIS
LIN {X -0.093,Y -289.885,Z 853.688,A 0.000,B 0.000,C 90.000,E1 303.833} C_DIS
LIN {X 0.062,Y -306.511,Z 853.669,A 0.000,B 0.000,C 90.000,E1 300.463} C_DIS
LIN {X 0.089,Y -319.360,Z 853.657,A 0.000,B 0.000,C 90.000,E1 298.180} C_DIS
LIN {X 0.008,Y -331.349,Z 853.646,A 0.000,B 0.000,C 90.000,E1 296.283} C_DIS
LIN {X -0.143,Y -350.880,Z 853.630,A 0.000,B 0.000,C 90.000,E1 293.515} C_DIS
LIN {X -0.088,Y -369.667,Z 853.617,A 0.000,B 0.000,C 90.000,E1 291.099} C_DIS
LIN {X -0.112,Y -395.349,Z 853.601,A 0.000,B 0.000,C 90.000,E1 288.236} C_DIS
LIN {X -0.173,Y -410.775,Z 853.592,A 0.000,B 0.000,C 90.000,E1 286.622} C_DIS
LIN {X -0.042,Y -420.815,Z 853.586,A 0.000,B 0.000,C 90.000,E1 285.552} C_DIS
LIN {X -0.248,Y -433.177,Z 853.579,A 0.000,B 0.000,C 90.000,E1 284.245} C_DIS
LIN {X 0.003,Y -445.073,Z 853.572,A 0.000,B 0.000,C 90.000,E1 282.883} C_DIS
LIN {X 0.062,Y -453.956,Z 853.566,A 0.000,B 0.000,C 90.000,E1 281.827} C_DIS
LIN {X 0.139,Y -462.303,Z 853.560,A 0.000,B 0.000,C 90.000,E1 280.782} C_DIS
LIN {X -0.139,Y -470.068,Z 853.554,A 0.000,B 0.000,C 90.000,E1 279.792} C_DIS
LIN {X -0.117,Y -475.380,Z 853.550,A 0.000,B 0.000,C 90.000,E1 279.029} C_DIS
LIN {X -0.133,Y -480.109,Z 853.546,A 0.000,B 0.000,C 90.000,E1 278.276} C_DIS
LIN {X -0.167,Y -484.165,Z 853.542,A 0.000,B 0.000,C 90.000,E1 277.530} C_DIS
LIN {X -0.103,Y -487.431,Z 853.538,A 0.000,B 0.000,C 90.000,E1 276.777} C_DIS
LIN {X 0.098,Y -489.202,Z 853.535,A 0.000,B 0.000,C 90.000,E1 276.258} C_DIS
LIN {X -0.180,Y -490.683,Z 853.532,A 0.000,B 0.000,C 90.000,E1 275.796} C_DIS
LIN {X 0.038,Y -491.787,Z 853.529,A 0.000,B 0.000,C 90.000,E1 275.277} C_DIS
LIN {X 0.263,Y -492.528,Z 853.527,A 0.000,B 0.000,C 90.000,E1 274.759} C_DIS
LIN {X -0.035,Y -492.900,Z 853.524,A 0.000,B 0.000,C 90.000,E1 274.302} C_DIS
LIN {X 0.200,Y -492.850,Z 853.521,A 0.000,B 0.000,C 90.000,E1 273.784} C_DIS
LIN {X -0.086,Y -492.449,Z 853.518,A 0.000,B 0.000,C 90.000,E1 273.326} C_DIS
LIN {X 0.147,Y -491.582,Z 853.516,A 0.000,B 0.000,C 90.000,E1 272.808} C_DIS
LIN {X -0.138,Y -490.285,Z 853.513,A 0.000,B 0.000,C 90.000,E1 272.350} C_DIS
LIN {X 0.066,Y -488.510,Z 853.510,A 0.000,B 0.000,C 90.000,E1 271.835} C_DIS
LIN {X -0.212,Y -486.195,Z 853.508,A 0.000,B 0.000,C 90.000,E1 271.375} C_DIS
LIN {X -0.033,Y -483.339,Z 853.505,A 0.000,B 0.000,C 90.000,E1 270.859} C_DIS
LIN {X 0.130,Y -479.746,Z 853.502,A 0.000,B 0.000,C 90.000,E1 270.344} C_DIS
LIN {X -0.203,Y -475.423,Z 853.499,A 0.000,B 0.000,C 90.000,E1 269.885} C_DIS
LIN {X -0.081,Y -470.170,Z 853.496,A 0.000,B 0.000,C 90.000,E1 269.370} C_DIS
LIN {X -0.125,Y -467.384,Z 853.495,A 0.000,B 0.000,C 90.000,E1 269.141} C_DIS
LIN {X 0.040,Y -461.185,Z 853.493,A 0.000,B 0.000,C 90.000,E1 268.682} C_DIS
LIN {X -0.211,Y -457.772,Z 853.492,A 0.000,B 0.000,C 90.000,E1 268.511} C_DIS
LIN {X -0.196,Y -450.546,Z 853.490,A 0.000,B 0.000,C 90.000,E1 268.165} C_DIS
LIN {X -0.070,Y -443.228,Z 853.488,A 0.000,B 0.000,C 90.000,E1 267.879} C_DIS
LIN {X 0.062,Y -435.352,Z 853.487,A 0.000,B 0.000,C 90.000,E1 267.650} C_DIS
LIN {X 0.181,Y -426.790,Z 853.486,A 0.000,B 0.000,C 90.000,E1 267.478} C_DIS
LIN {X 0.003,Y -419.570,Z 853.486,A 0.000,B 0.000,C 90.000,E1 267.421} C_DIS
LIN {X 0.166,Y -412.158,Z 853.485,A 0.000,B 0.000,C 90.000,E1 267.364} C_DIS
LIN {X 0.049,Y -181.035,Z 853.485,A 0.000,B 0.000,C 90.000,E1 267.364} C_DIS
LIN {X 0.081,Y -180.807,Z 853.471,A 0.000,B 0.000,C 90.000,E1 264.780} C_DIS
LIN {X -0.022,Y -178.908,Z 853.443,A 0.000,B 0.000,C 90.000,E1 259.746} C_DIS
LIN {X 0.059,Y -175.952,Z 853.415,A 0.000,B 0.000,C 90.000,E1 254.629} C_DIS
LIN {X 0.005,Y -175.417,Z 853.410,A 0.000,B 0.000,C 90.000,E1 253.795} C_DIS
LIN {X 0.008,Y -172.180,Z 853.386,A 0.000,B 0.000,C 90.000,E1 249.518} C_DIS
LIN {X 0.047,Y -171.652,Z 853.381,A 0.000,B 0.000,C 90.000,E1 248.646} C_DIS
LIN {X 0.042,Y -167.875,Z 853.357,A 0.000,B 0.000,C 90.000,E1 244.332} C_DIS
LIN {X -0.016,Y -166.610,Z 853.348,A 0.000,B 0.000,C 90.000,E1 242.615} C_DIS
LIN {X -0.021,Y -162.598,Z 853.324,A 0.000,B 0.000,C 90.000,E1 238.250} C_DIS
LIN {X -0.047,Y -161.283,Z 853.314,A 0.000,B 0.000,C 90.000,E1 236.501} C_DIS
LIN {X -0.012,Y -157.282,Z 853.289,A 0.000,B 0.000,C 90.000,E1 232.065} C_DIS
LIN {X 0.010,Y -156.000,Z 853.279,A 0.000,B 0.000,C 90.000,E1 230.275} C_DIS
LIN {X -0.029,Y -152.258,Z 853.254,A 0.000,B 0.000,C 90.000,E1 225.810} C_DIS
LIN {X -0.007,Y -150.496,Z 853.239,A 0.000,B 0.000,C 90.000,E1 223.095} C_DIS
LIN {X 0.023,Y -147.220,Z 853.214,A 0.000,B 0.000,C 90.000,E1 218.543} C_DIS
LIN {X -0.007,Y -145.243,Z 853.194,A 0.000,B 0.000,C 90.000,E1 214.898} C_DIS
LIN {X -0.091,Y -142.362,Z 853.163,A 0.000,B 0.000,C 90.000,E1 209.411} C_DIS
LIN {X 0.030,Y -141.748,Z 853.153,A 0.000,B 0.000,C 90.000,E1 207.513} C_DIS
LIN {X -0.043,Y -139.492,Z 853.117,A 0.000,B 0.000,C 90.000,E1 201.046} C_DIS
LIN {X -0.007,Y -138.996,Z 853.101,A 0.000,B 0.000,C 90.000,E1 198.236} C_DIS
LIN {X -0.051,Y -138.337,Z 853.055,A 0.000,B 0.000,C 90.000,E1 189.849} C_DIS
LIN {X -0.028,Y -139.414,Z 853.008,A 0.000,B 0.000,C 90.000,E1 181.432} C_DIS
LIN {X 0.025,Y -141.328,Z 852.972,A 0.000,B 0.000,C 90.000,E1 174.894} C_DIS
LIN {X -0.018,Y -142.686,Z 852.956,A 0.000,B 0.000,C 90.000,E1 172.129} C_DIS
LIN {X -0.038,Y -145.045,Z 852.931,A 0.000,B 0.000,C 90.000,E1 167.521} C_DIS
LIN {X -0.041,Y -147.671,Z 852.910,A 0.000,B 0.000,C 90.000,E1 163.850} C_DIS
LIN {X -0.006,Y -150.313,Z 852.890,A 0.000,B 0.000,C 90.000,E1 160.188} C_DIS
LIN {X 0.066,Y -153.726,Z 852.870,A 0.000,B 0.000,C 90.000,E1 156.538} C_DIS
LIN {X -0.083,Y -157.139,Z 852.850,A 0.000,B 0.000,C 90.000,E1 152.999} C_DIS
LIN {X -0.007,Y -161.288,Z 852.830,A 0.000,B 0.000,C 90.000,E1 149.410} C_DIS
LIN {X 0.010,Y -164.404,Z 852.815,A 0.000,B 0.000,C 90.000,E1 146.755} C_DIS
LIN {X 0.007,Y -169.084,Z 852.796,A 0.000,B 0.000,C 90.000,E1 143.256} C_DIS
LIN {X -0.043,Y -171.642,Z 852.786,A 0.000,B 0.000,C 90.000,E1 141.537} C_DIS
LIN {X 0.004,Y -176.603,Z 852.767,A 0.000,B 0.000,C 90.000,E1 138.081} C_DIS
LIN {X 0.005,Y -180.901,Z 852.753,A 0.000,B 0.000,C 90.000,E1 135.526} C_DIS
LIN {X -0.003,Y -186.317,Z 852.734,A 0.000,B 0.000,C 90.000,E1 132.162} C_DIS
LIN {X 0.063,Y -190.951,Z 852.720,A 0.000,B 0.000,C 90.000,E1 129.644} C_DIS
LIN {X -0.086,Y -192.985,Z 852.714,A 0.000,B 0.000,C 90.000,E1 128.463} C_DIS
LIN {X -0.165,Y -293.475,Z 852.714,A 0.000,B 0.000,C 90.000,E1 128.463} C_DIS
LIN {X 0.008,Y -296.140,Z 852.713,A 0.000,B 0.000,C 90.000,E1 128.382} C_DIS
LIN {X 0.114,Y -299.904,Z 852.712,A 0.000,B 0.000,C 90.000,E1 128.177} C_DIS
LIN {X -0.016,Y -302.161,Z 852.711,A 0.000,B 0.000,C 90.000,E1 128.016} C_DIS
LIN {X 0.032,Y -306.022,Z 852.708,A 0.000,B 0.000,C 90.000,E1 127.523} C_DIS
LIN {X -0.013,Y -307.841,Z 852.707,A 0.000,B 0.000,C 90.000,E1 127.202} C_DIS
LIN {X 0.001,Y -309.261,Z 852.705,A 0.000,B 0.000,C 90.000,E1 126.870} C_DIS
LIN {X 0.003,Y -311.307,Z 852.701,A 0.000,B 0.000,C 90.000,E1 126.217} C_DIS
LIN {X 0.172,Y -321.507,Z 852.683,A 0.000,B 0.000,C 90.000,E1 122.959} C_DIS
LIN {X 0.052,Y -332.013,Z 852.667,A 0.000,B 0.000,C 90.000,E1 120.129} C_DIS
LIN {X 0.020,Y -343.879,Z 852.652,A 0.000,B 0.000,C 90.000,E1 117.334} C_DIS
LIN {X 0.025,Y -357.207,Z 852.637,A 0.000,B 0.000,C 90.000,E1 114.591} C_DIS
LIN {X 0.017,Y -370.378,Z 852.623,A 0.000,B 0.000,C 90.000,E1 112.206} C_DIS
LIN {X -0.081,Y -384.894,Z 852.610,A 0.000,B 0.000,C 90.000,E1 109.885} C_DIS
LIN {X 0.060,Y -400.858,Z 852.598,A 0.000,B 0.000,C 90.000,E1 107.583} C_DIS
LIN {X -0.027,Y -418.385,Z 852.585,A 0.000,B 0.000,C 90.000,E1 105.371} C_DIS
LIN {X 0.226,Y -437.571,Z 852.573,A 0.000,B 0.000,C 90.000,E1 103.175} C_DIS
LIN {X -0.015,Y -457.720,Z 852.562,A 0.000,B 0.000,C 90.000,E1 101.186} C_DIS
LIN {X -0.129,Y -467.907,Z 852.557,A 0.000,B 0.000,C 90.000,E1 100.254} C_DIS
LIN {X -0.097,Y -469.831,Z 852.556,A 0.000,B 0.000,C 90.000,E1 100.018} C_DIS
LIN {X 0.216,Y -471.425,Z 852.554,A 0.000,B 0.000,C 90.000,E1 99.726} C_DIS
LIN {X -0.013,Y -472.622,Z 852.553,A 0.000,B 0.000,C 90.000,E1 99.500} C_DIS
LIN {X 0.169,Y -474.078,Z 852.550,A 0.000,B 0.000,C 90.000,E1 98.973} C_DIS
LIN {X -0.186,Y -474.501,Z 852.547,A 0.000,B 0.000,C 90.000,E1 98.511} C_DIS
LIN {X -0.060,Y -473.962,Z 852.544,A 0.000,B 0.000,C 90.000,E1 97.992} C_DIS
LIN {X 0.069,Y -472.380,Z 852.542,A 0.000,B 0.000,C 90.000,E1 97.473} C_DIS
LIN {X -0.073,Y -471.113,Z 852.540,A 0.000,B 0.000,C 90.000,E1 97.239} C_DIS
LIN {X -0.137,Y -454.966,Z 852.526,A 0.000,B 0.000,C 90.000,E1 94.702} C_DIS
LIN {X 0.031,Y -444.418,Z 852.516,A 0.000,B 0.000,C 90.000,E1 92.865} C_DIS
LIN {X -0.202,Y -435.150,Z 852.507,A 0.000,B 0.000,C 90.000,E1 91.318} C_DIS
LIN {X -0.164,Y -425.562,Z 852.498,A 0.000,B 0.000,C 90.000,E1 89.714} C_DIS
LIN {X -0.088,Y -412.528,Z 852.486,A 0.000,B 0.000,C 90.000,E1 87.535} C_DIS
LIN {X -0.003,Y -402.688,Z 852.477,A 0.000,B 0.000,C 90.000,E1 85.869} C_DIS
LIN {X -0.037,Y -391.265,Z 852.466,A 0.000,B 0.000,C 90.000,E1 83.913} C_DIS
LIN {X 0.118,Y -380.050,Z 852.455,A 0.000,B 0.000,C 90.000,E1 81.894} C_DIS
LIN {X 0.051,Y -365.859,Z 852.440,A 0.000,B 0.000,C 90.000,E1 79.285} C_DIS
LIN {X -0.130,Y -353.628,Z 852.427,A 0.000,B 0.000,C 90.000,E1 76.937} C_DIS
LIN {X -0.083,Y -342.852,Z 852.416,A 0.000,B 0.000,C 90.000,E1 74.810} C_DIS
LIN {X 0.081,Y -329.230,Z 852.400,A 0.000,B 0.000,C 90.000,E1 72.000} C_DIS
LIN {X 0.066,Y -316.096,Z 852.384,A 0.000,B 0.000,C 90.000,E1 69.156} C_DIS
LIN {X 0.137,Y -303.367,Z 852.368,A 0.000,B 0.000,C 90.000,E1 66.230} C_DIS
LIN {X -0.147,Y -292.368,Z 852.353,A 0.000,B 0.000,C 90.000,E1 63.640} C_DIS
LIN {X -0.012,Y -282.950,Z 852.340,A 0.000,B 0.000,C 90.000,E1 61.257} C_DIS
LIN {X 0.047,Y -271.062,Z 852.323,A 0.000,B 0.000,C 90.000,E1 58.152} C_DIS
LIN {X 0.018,Y -258.685,Z 852.304,A 0.000,B 0.000,C 90.000,E1 54.642} C_DIS
LIN {X 0.006,Y -247.333,Z 852.284,A 0.000,B 0.000,C 90.000,E1 51.045} C_DIS
LIN {X -0.057,Y -237.932,Z 852.265,A 0.000,B 0.000,C 90.000,E1 47.757} C_DIS
LIN {X -0.102,Y -228.209,Z 852.244,A 0.000,B 0.000,C 90.000,E1 44.028} C_DIS
LIN {X 0.052,Y -219.186,Z 852.223,A 0.000,B 0.000,C 90.000,E1 40.172} C_DIS
LIN {X 0.004,Y -210.651,Z 852.202,A 0.000,B 0.000,C 90.000,E1 36.297} C_DIS
LIN {X -0.104,Y -204.293,Z 852.184,A 0.000,B 0.000,C 90.000,E1 33.166} C_DIS
LIN {X 0.032,Y -198.474,Z 852.166,A 0.000,B 0.000,C 90.000,E1 29.922} C_DIS
LIN {X -0.024,Y -193.295,Z 852.148,A 0.000,B 0.000,C 90.000,E1 26.693} C_DIS
LIN {X 0.055,Y -188.829,Z 852.130,A 0.000,B 0.000,C 90.000,E1 23.387} C_DIS
LIN {X 0.071,Y -185.182,Z 852.112,A 0.000,B 0.000,C 90.000,E1 20.066} C_DIS
LIN {X 0.029,Y -181.649,Z 852.088,A 0.000,B 0.000,C 90.000,E1 15.898} C_DIS
LIN {X 0.036,Y -178.952,Z 852.060,A 0.000,B 0.000,C 90.000,E1 10.838} C_DIS
LIN {X -0.019,Y -179.610,Z 851.974,A 0.000,B 0.000,C 90.000,E1 355.298} C_DIS
LIN {X 0.062,Y -182.740,Z 851.946,A 0.000,B 0.000,C 90.000,E1 350.208} C_DIS
LIN {X -0.034,Y -186.450,Z 851.922,A 0.000,B 0.000,C 90.000,E1 346.047} C_DIS
LIN {X -0.045,Y -190.142,Z 851.904,A 0.000,B 0.000,C 90.000,E1 342.725} C_DIS
LIN {X 0.004,Y -195.594,Z 851.881,A 0.000,B 0.000,C 90.000,E1 338.592} C_DIS
LIN {X -0.032,Y -201.934,Z 851.858,A 0.000,B 0.000,C 90.000,E1 334.537} C_DIS
LIN {X -0.072,Y -209.062,Z 851.836,A 0.000,B 0.000,C 90.000,E1 330.539} C_DIS
LIN {X -0.022,Y -216.875,Z 851.814,A 0.000,B 0.000,C 90.000,E1 326.580} C_DIS
LIN {X 0.011,Y -223.732,Z 851.797,A 0.000,B 0.000,C 90.000,E1 323.463} C_DIS
LIN {X -0.042,Y -232.343,Z 851.778,A 0.000,B 0.000,C 90.000,E1 320.033} C_DIS
LIN {X -0.062,Y -241.818,Z 851.759,A 0.000,B 0.000,C 90.000,E1 316.662} C_DIS
LIN {X 0.007,Y -252.276,Z 851.741,A 0.000,B 0.000,C 90.000,E1 313.338} C_DIS
LIN {X 0.041,Y -263.792,Z 851.723,A 0.000,B 0.000,C 90.000,E1 310.092} C_DIS
LIN {X -0.069,Y -276.272,Z 851.705,A 0.000,B 0.000,C 90.000,E1 306.950} C_DIS
LIN {X 0.065,Y -289.930,Z 851.688,A 0.000,B 0.000,C 90.000,E1 303.833} C_DIS
LIN {X -0.055,Y -304.758,Z 851.671,A 0.000,B 0.000,C 90.000,E1 300.846} C_DIS
LIN {X 0.013,Y -315.481,Z 851.660,A 0.000,B 0.000,C 90.000,E1 298.871} C_DIS
LIN {X 0.040,Y -331.143,Z 851.646,A 0.000,B 0.000,C 90.000,E1 296.309} C_DIS
LIN {X 0.029,Y -348.389,Z 851.632,A 0.000,B 0.000,C 90.000,E1 293.823} C_DIS
LIN {X -0.047,Y -364.442,Z 851.621,A 0.000,B 0.000,C 90.000,E1 291.716} C_DIS
LIN {X -0.133,Y -384.475,Z 851.608,A 0.000,B 0.000,C 90.000,E1 289.396} C_DIS
LIN {X 0.208,Y -399.878,Z 851.598,A 0.000,B 0.000,C 90.000,E1 287.692} C_DIS
LIN {X 0.155,Y -415.346,Z 851.589,A 0.000,B 0.000,C 90.000,E1 286.079} C_DIS
LIN {X -0.123,Y -425.261,Z 851.584,A 0.000,B 0.000,C 90.000,E1 285.064} C_DIS
LIN {X 0.022,Y -437.569,Z 851.576,A 0.000,B 0.000,C 90.000,E1 283.703} C_DIS
LIN {X -0.010,Y -446.950,Z 851.570,A 0.000,B 0.000,C 90.000,E1 282.647} C_DIS
LIN {X 0.069,Y -455.756,Z 851.564,A 0.000,B 0.000,C 90.000,E1 281.591} C_DIS
LIN {X 0.167,Y -463.975,Z 851.559,A 0.000,B 0.000,C 90.000,E1 280.546} C_DIS
LIN {X 0.056,Y -469.750,Z 851.554,A 0.000,B 0.000,C 90.000,E1 279.792} C_DIS
LIN {X 0.078,Y -475.113,Z 851.550,A 0.000,B 0.000,C 90.000,E1 279.029} C_DIS
LIN {X 0.062,Y -479.880,Z 851.546,A 0.000,B 0.000,C 90.000,E1 278.276} C_DIS
LIN {X 0.026,Y -483.977,Z 851.542,A 0.000,B 0.000,C 90.000,E1 277.530} C_DIS
LIN {X 0.090,Y -487.271,Z 851.538,A 0.000,B 0.000,C 90.000,E1 276.777} C_DIS
LIN {X -0.195,Y -489.056,Z 851.535,A 0.000,B 0.000,C 90.000,E1 276.315} C_DIS
LIN {X 0.013,Y -490.564,Z 851.532,A 0.000,B 0.000,C 90.000,E1 275.796} C_DIS
LIN {X 0.230,Y -491.689,Z 851.529,A 0.000,B 0.000,C 90.000,E1 275.277} C_DIS
LIN {X -0.077,Y -492.423,Z 851.527,A 0.000,B 0.000,C 90.000,E1 274.821} C_DIS
LIN {X 0.156,Y -492.833,Z 851.524,A 0.000,B 0.000,C 90.000,E1 274.302} C_DIS
LIN {X -0.100,Y -492.850,Z 851.521,A 0.000,B 0.000,C 90.000,E1 273.841} C_DIS
LIN {X 0.104,Y -492.460,Z 851.519,A 0.000,B 0.000,C 90.000,E1 273.326} C_DIS
LIN {X -0.154,Y -491.637,Z 851.516,A 0.000,B 0.000,C 90.000,E1 272.865} C_DIS
LIN {X 0.052,Y -490.383,Z 851.513,A 0.000,B 0.000,C 90.000,E1 272.350} C_DIS
LIN {X -0.234,Y -488.672,Z 851.510,A 0.000,B 0.000,C 90.000,E1 271.892} C_DIS
LIN {X -0.023,Y -486.436,Z 851.508,A 0.000,B 0.000,C 90.000,E1 271.375} C_DIS
LIN {X 0.155,Y -483.630,Z 851.505,A 0.000,B 0.000,C 90.000,E1 270.859} C_DIS
LIN {X -0.161,Y -480.134,Z 851.502,A 0.000,B 0.000,C 90.000,E1 270.401} C_DIS
LIN {X -0.014,Y -475.907,Z 851.499,A 0.000,B 0.000,C 90.000,E1 269.885} C_DIS
LIN {X 0.109,Y -470.803,Z 851.497,A 0.000,B 0.000,C 90.000,E1 269.370} C_DIS
LIN {X -0.035,Y -464.889,Z 851.494,A 0.000,B 0.000,C 90.000,E1 268.912} C_DIS
LIN {X 0.120,Y -461.829,Z 851.493,A 0.000,B 0.000,C 90.000,E1 268.682} C_DIS
LIN {X -0.195,Y -455.052,Z 851.491,A 0.000,B 0.000,C 90.000,E1 268.339} C_DIS
LIN {X 0.073,Y -447.888,Z 851.489,A 0.000,B 0.000,C 90.000,E1 267.993} C_DIS
LIN {X -0.052,Y -440.422,Z 851.488,A 0.000,B 0.000,C 90.000,E1 267.764} C_DIS
LIN {X -0.177,Y -432.265,Z 851.487,A 0.000,B 0.000,C 90.000,E1 267.593} C_DIS
LIN {X 0.086,Y -422.896,Z 851.486,A 0.000,B 0.000,C 90.000,E1 267.421} C_DIS
LIN {X 0.042,Y -413.669,Z 851.485,A 0.000,B 0.000,C 90.000,E1 267.364} C_DIS
LIN {X -0.006,Y -181.033,Z 851.485,A 0.000,B 0.000,C 90.000,E1 267.364} C_DIS
LIN {X 0.022,Y -180.800,Z 851.471,A 0.000,B 0.000,C 90.000,E1 264.780} C_DIS
LIN {X -0.080,Y -178.900,Z 851.443,A 0.000,B 0.000,C 90.000,E1 259.746} C_DIS
LIN {X 0.000,Y -175.943,Z 851.415,A 0.000,B 0.000,C 90.000,E1 254.629} C_DIS
LIN {X -0.053,Y -175.401,Z 851.410,A 0.000,B 0.000,C 90.000,E1 253.795} C_DIS
LIN {X -0.049,Y -172.169,Z 851.386,A 0.000,B 0.000,C 90.000,E1 249.518} C_DIS
LIN {X -0.010,Y -171.637,Z 851.381,A 0.000,B 0.000,C 90.000,E1 248.646} C_DIS
LIN {X -0.015,Y -167.861,Z 851.357,A 0.000,B 0.000,C 90.000,E1 244.332} C_DIS
LIN {X -0.072,Y -166.593,Z 851.348,A 0.000,B 0.000,C 90.000,E1 242.615} C_DIS
LIN {X 0.062,Y -162.583,Z 851.323,A 0.000,B 0.000,C 90.000,E1 238.201} C_DIS
LIN {X -0.103,Y -161.266,Z 851.314,A 0.000,B 0.000,C 90.000,E1 236.501} C_DIS
LIN {X 0.030,Y -157.267,Z 851.289,A 0.000,B 0.000,C 90.000,E1 232.029} C_DIS
LIN {X -0.044,Y -155.987,Z 851.279,A 0.000,B 0.000,C 90.000,E1 230.275} C_DIS
LIN {X -0.082,Y -152.244,Z 851.254,A 0.000,B 0.000,C 90.000,E1 225.810} C_DIS
LIN {X -0.060,Y -150.484,Z 851.239,A 0.000,B 0.000,C 90.000,E1 223.095} C_DIS
LIN {X -0.029,Y -147.208,Z 851.214,A 0.000,B 0.000,C 90.000,E1 218.543} C_DIS
LIN {X -0.059,Y -145.229,Z 851.194,A 0.000,B 0.000,C 90.000,E1 214.898} C_DIS
LIN {X 0.052,Y -142.354,Z 851.163,A 0.000,B 0.000,C 90.000,E1 209.333} C_DIS
LIN {X -0.021,Y -141.741,Z 851.153,A 0.000,B 0.000,C 90.000,E1 207.513} C_DIS
LIN {X 0.086,Y -139.488,Z 851.117,A 0.000,B 0.000,C 90.000,E1 200.972} C_DIS
LIN {X -0.057,Y -138.991,Z 851.101,A 0.000,B 0.000,C 90.000,E1 198.236} C_DIS
LIN {X 0.036,Y -138.336,Z 851.055,A 0.000,B 0.000,C 90.000,E1 189.792} C_DIS
LIN {X 0.060,Y -139.419,Z 851.008,A 0.000,B 0.000,C 90.000,E1 181.375} C_DIS
LIN {X -0.026,Y -141.337,Z 850.972,A 0.000,B 0.000,C 90.000,E1 174.894} C_DIS
LIN {X -0.069,Y -142.694,Z 850.956,A 0.000,B 0.000,C 90.000,E1 172.129} C_DIS
LIN {X 0.052,Y -145.058,Z 850.930,A 0.000,B 0.000,C 90.000,E1 167.465} C_DIS
LIN {X 0.049,Y -147.683,Z 850.910,A 0.000,B 0.000,C 90.000,E1 163.795} C_DIS
LIN {X -0.059,Y -150.330,Z 850.890,A 0.000,B 0.000,C 90.000,E1 160.188} C_DIS
LIN {X 0.012,Y -153.747,Z 850.870,A 0.000,B 0.000,C 90.000,E1 156.538} C_DIS
LIN {X 0.003,Y -157.161,Z 850.850,A 0.000,B 0.000,C 90.000,E1 152.948} C_DIS
LIN {X -0.063,Y -161.313,Z 850.830,A 0.000,B 0.000,C 90.000,E1 149.410} C_DIS
LIN {X -0.046,Y -164.427,Z 850.815,A 0.000,B 0.000,C 90.000,E1 146.755} C_DIS
LIN {X -0.050,Y -169.113,Z 850.796,A 0.000,B 0.000,C 90.000,E1 143.256} C_DIS
LIN {X -0.099,Y -171.667,Z 850.786,A 0.000,B 0.000,C 90.000,E1 141.537} C_DIS
LIN {X -0.054,Y -176.634,Z 850.767,A 0.000,B 0.000,C 90.000,E1 138.081} C_DIS
LIN {X 0.073,Y -180.931,Z 850.753,A 0.000,B 0.000,C 90.000,E1 135.486} C_DIS
LIN {X -0.064,Y -186.350,Z 850.734,A 0.000,B 0.000,C 90.000,E1 132.162} C_DIS
LIN {X 0.002,Y -190.982,Z 850.720,A 0.000,B 0.000,C 90.000,E1 129.644} C_DIS
LIN {X -0.063,Y -192.973,Z 850.714,A 0.000,B 0.000,C 90.000,E1 128.463} C_DIS
LIN {X -0.138,Y -293.731,Z 850.714,A 0.000,B 0.000,C 90.000,E1 128.463} C_DIS
LIN {X 0.008,Y -294.960,Z 850.713,A 0.000,B 0.000,C 90.000,E1 128.418} C_DIS
LIN {X -0.076,Y -299.841,Z 850.712,A 0.000,B 0.000,C 90.000,E1 128.222} C_DIS
LIN {X -0.113,Y -302.378,Z 850.711,A 0.000,B 0.000,C 90.000,E1 128.016} C_DIS
LIN {X -0.105,Y -306.184,Z 850.708,A 0.000,B 0.000,C 90.000,E1 127.523} C_DIS
LIN {X 0.095,Y -307.957,Z 850.707,A 0.000,B 0.000,C 90.000,E1 127.156} C_DIS
LIN {X -0.136,Y -309.342,Z 850.705,A 0.000,B 0.000,C 90.000,E1 126.870} C_DIS
LIN {X 0.072,Y -318.354,Z 850.688,A 0.000,B 0.000,C 90.000,E1 123.913} C_DIS
LIN {X 0.025,Y -328.441,Z 850.673,A 0.000,B 0.000,C 90.000,E1 121.052} C_DIS
LIN {X 0.050,Y -339.854,Z 850.657,A 0.000,B 0.000,C 90.000,E1 118.231} C_DIS
LIN {X 0.085,Y -352.697,Z 850.642,A 0.000,B 0.000,C 90.000,E1 115.463} C_DIS
LIN {X -0.038,Y -365.403,Z 850.628,A 0.000,B 0.000,C 90.000,E1 113.078} C_DIS
LIN {X -0.127,Y -379.418,Z 850.615,A 0.000,B 0.000,C 90.000,E1 110.737} C_DIS
LIN {X -0.002,Y -394.842,Z 850.602,A 0.000,B 0.000,C 90.000,E1 108.417} C_DIS
LIN {X -0.247,Y -411.785,Z 850.590,A 0.000,B 0.000,C 90.000,E1 106.205} C_DIS
LIN {X -0.190,Y -430.370,Z 850.578,A 0.000,B 0.000,C 90.000,E1 104.008} C_DIS
LIN {X 0.127,Y -450.297,Z 850.566,A 0.000,B 0.000,C 90.000,E1 101.883} C_DIS
LIN {X 0.169,Y -468.074,Z 850.557,A 0.000,B 0.000,C 90.000,E1 100.197} C_DIS
LIN {X 0.205,Y -469.963,Z 850.555,A 0.000,B 0.000,C 90.000,E1 99.962} C_DIS
LIN {X 0.055,Y -471.533,Z 850.554,A 0.000,B 0.000,C 90.000,E1 99.726} C_DIS
LIN {X -0.175,Y -472.708,Z 850.553,A 0.000,B 0.000,C 90.000,E1 99.500} C_DIS
LIN {X 0.008,Y -474.133,Z 850.550,A 0.000,B 0.000,C 90.000,E1 98.973} C_DIS
LIN {X 0.123,Y -474.530,Z 850.547,A 0.000,B 0.000,C 90.000,E1 98.454} C_DIS
LIN {X -0.221,Y -473.963,Z 850.544,A 0.000,B 0.000,C 90.000,E1 97.992} C_DIS
LIN {X -0.029,Y -472.349,Z 850.541,A 0.000,B 0.000,C 90.000,E1 97.466} C_DIS
LIN {X -0.231,Y -471.060,Z 850.540,A 0.000,B 0.000,C 90.000,E1 97.239} C_DIS
LIN {X 0.161,Y -454.886,Z 850.526,A 0.000,B 0.000,C 90.000,E1 94.645} C_DIS
LIN {X -0.123,Y -444.343,Z 850.516,A 0.000,B 0.000,C 90.000,E1 92.865} C_DIS
LIN {X 0.082,Y -435.064,Z 850.507,A 0.000,B 0.000,C 90.000,E1 91.260} C_DIS
LIN {X 0.113,Y -425.469,Z 850.498,A 0.000,B 0.000,C 90.000,E1 89.656} C_DIS
LIN {X 0.177,Y -412.422,Z 850.486,A 0.000,B 0.000,C 90.000,E1 87.478} C_DIS
LIN {X -0.148,Y -402.582,Z 850.477,A 0.000,B 0.000,C 90.000,E1 85.869} C_DIS
LIN {X -0.181,Y -391.167,Z 850.466,A 0.000,B 0.000,C 90.000,E1 83.913} C_DIS
LIN {X -0.001,Y -378.343,Z 850.453,A 0.000,B 0.000,C 90.000,E1 81.602} C_DIS
LIN {X -0.103,Y -364.213,Z 850.439,A 0.000,B 0.000,C 90.000,E1 78.993} C_DIS
LIN {X 0.027,Y -352.042,Z 850.426,A 0.000,B 0.000,C 90.000,E1 76.589} C_DIS
LIN {X 0.115,Y -341.264,Z 850.414,A 0.000,B 0.000,C 90.000,E1 74.448} C_DIS
LIN {X -0.075,Y -327.759,Z 850.398,A 0.000,B 0.000,C 90.000,E1 71.692} C_DIS
LIN {X 0.056,Y -316.109,Z 850.384,A 0.000,B 0.000,C 90.000,E1 69.135} C_DIS
LIN {X 0.018,Y -303.398,Z 850.368,A 0.000,B 0.000,C 90.000,E1 66.230} C_DIS
LIN {X 0.137,Y -293.792,Z 850.355,A 0.000,B 0.000,C 90.000,E1 63.896} C_DIS
LIN {X 0.040,Y -284.400,Z 850.342,A 0.000,B 0.000,C 90.000,E1 61.563} C_DIS
LIN {X 0.067,Y -273.806,Z 850.327,A 0.000,B 0.000,C 90.000,E1 58.820} C_DIS
LIN {X -0.023,Y -261.345,Z 850.307,A 0.000,B 0.000,C 90.000,E1 55.341} C_DIS
LIN {X 0.052,Y -249.837,Z 850.288,A 0.000,B 0.000,C 90.000,E1 51.743} C_DIS
LIN {X -0.073,Y -240.263,Z 850.269,A 0.000,B 0.000,C 90.000,E1 48.485} C_DIS
LIN {X -0.051,Y -230.412,Z 850.249,A 0.000,B 0.000,C 90.000,E1 44.757} C_DIS
LIN {X 0.008,Y -221.267,Z 850.227,A 0.000,B 0.000,C 90.000,E1 40.943} C_DIS
LIN {X -0.007,Y -212.614,Z 850.206,A 0.000,B 0.000,C 90.000,E1 37.076} C_DIS
LIN {X -0.120,Y -204.586,Z 850.184,A 0.000,B 0.000,C 90.000,E1 33.166} C_DIS
LIN {X 0.022,Y -198.777,Z 850.166,A 0.000,B 0.000,C 90.000,E1 29.922} C_DIS
LIN {X -0.026,Y -193.592,Z 850.148,A 0.000,B 0.000,C 90.000,E1 26.693} C_DIS
LIN {X 0.061,Y -189.115,Z 850.130,A 0.000,B 0.000,C 90.000,E1 23.387} C_DIS
LIN {X -0.090,Y -185.476,Z 850.112,A 0.000,B 0.000,C 90.000,E1 20.120} C_DIS
LIN {X 0.051,Y -181.960,Z 850.088,A 0.000,B 0.000,C 90.000,E1 15.898} C_DIS
LIN {X 0.069,Y -179.271,Z 850.060,A 0.000,B 0.000,C 90.000,E1 10.838} C_DIS
LIN {X -0.010,Y -179.947,Z 849.974,A 0.000,B 0.000,C 90.000,E1 355.298} C_DIS
LIN {X 0.054,Y -183.078,Z 849.946,A 0.000,B 0.000,C 90.000,E1 350.218} C_DIS
LIN {X 0.001,Y -186.775,Z 849.922,A 0.000,B 0.000,C 90.000,E1 346.047} C_DIS
LIN {X -0.003,Y -190.466,Z 849.904,A 0.000,B 0.000,C 90.000,E1 342.725} C_DIS
LIN {X 0.059,Y -195.896,Z 849.881,A 0.000,B 0.000,C 90.000,E1 338.592} C_DIS
LIN {X 0.033,Y -202.219,Z 849.859,A 0.000,B 0.000,C 90.000,E1 334.537} C_DIS
LIN {X 0.004,Y -209.322,Z 849.836,A 0.000,B 0.000,C 90.000,E1 330.539} C_DIS
LIN {X 0.066,Y -217.118,Z 849.814,A 0.000,B 0.000,C 90.000,E1 326.580} C_DIS
LIN {X -0.026,Y -223.953,Z 849.797,A 0.000,B 0.000,C 90.000,E1 323.497} C_DIS
LIN {X -0.084,Y -232.556,Z 849.778,A 0.000,B 0.000,C 90.000,E1 320.070} C_DIS
LIN {X 0.055,Y -242.012,Z 849.759,A 0.000,B 0.000,C 90.000,E1 316.662} C_DIS
LIN {X -0.049,Y -252.450,Z 849.741,A 0.000,B 0.000,C 90.000,E1 313.380} C_DIS
LIN {X -0.022,Y -263.929,Z 849.723,A 0.000,B 0.000,C 90.000,E1 310.135} C_DIS
LIN {X 0.079,Y -276.340,Z 849.705,A 0.000,B 0.000,C 90.000,E1 306.950} C_DIS
LIN {X 0.060,Y -289.968,Z 849.688,A 0.000,B 0.000,C 90.000,E1 303.865} C_DIS
LIN {X -0.046,Y -304.728,Z 849.672,A 0.000,B 0.000,C 90.000,E1 300.875} C_DIS
LIN {X 0.031,Y -315.398,Z 849.661,A 0.000,B 0.000,C 90.000,E1 298.899} C_DIS
LIN {X -0.080,Y -330.983,Z 849.646,A 0.000,B 0.000,C 90.000,E1 296.360} C_DIS
LIN {X -0.100,Y -350.335,Z 849.631,A 0.000,B 0.000,C 90.000,E1 293.567} C_DIS
LIN {X -0.067,Y -368.952,Z 849.617,A 0.000,B 0.000,C 90.000,E1 291.153} C_DIS
LIN {X -0.112,Y -391.682,Z 849.603,A 0.000,B 0.000,C 90.000,E1 288.598} C_DIS
LIN {X -0.011,Y -409.656,Z 849.593,A 0.000,B 0.000,C 90.000,E1 286.677} C_DIS
LIN {X -0.016,Y -419.851,Z 849.587,A 0.000,B 0.000,C 90.000,E1 285.607} C_DIS
LIN {X 0.186,Y -432.229,Z 849.579,A 0.000,B 0.000,C 90.000,E1 284.245} C_DIS
LIN {X -0.150,Y -441.797,Z 849.573,A 0.000,B 0.000,C 90.000,E1 283.231} C_DIS
LIN {X -0.136,Y -450.955,Z 849.568,A 0.000,B 0.000,C 90.000,E1 282.175} C_DIS
LIN {X -0.102,Y -459.493,Z 849.562,A 0.000,B 0.000,C 90.000,E1 281.130} C_DIS
LIN {X 0.125,Y -467.480,Z 849.556,A 0.000,B 0.000,C 90.000,E1 280.074} C_DIS
LIN {X -0.178,Y -474.768,Z 849.550,A 0.000,B 0.000,C 90.000,E1 279.095} C_DIS
LIN {X -0.195,Y -479.590,Z 849.546,A 0.000,B 0.000,C 90.000,E1 278.341} C_DIS
LIN {X -0.166,Y -483.716,Z 849.542,A 0.000,B 0.000,C 90.000,E1 277.587} C_DIS
LIN {X -0.106,Y -487.040,Z 849.538,A 0.000,B 0.000,C 90.000,E1 276.834} C_DIS
LIN {X 0.093,Y -488.868,Z 849.535,A 0.000,B 0.000,C 90.000,E1 276.315} C_DIS
LIN {X -0.189,Y -490.411,Z 849.532,A 0.000,B 0.000,C 90.000,E1 275.853} C_DIS
LIN {X 0.027,Y -491.556,Z 849.530,A 0.000,B 0.000,C 90.000,E1 275.334} C_DIS
LIN {X 0.209,Y -492.314,Z 849.527,A 0.000,B 0.000,C 90.000,E1 274.821} C_DIS
LIN {X -0.050,Y -492.760,Z 849.524,A 0.000,B 0.000,C 90.000,E1 274.359} C_DIS
LIN {X 0.185,Y -492.820,Z 849.521,A 0.000,B 0.000,C 90.000,E1 273.841} C_DIS
LIN {X -0.103,Y -492.470,Z 849.519,A 0.000,B 0.000,C 90.000,E1 273.383} C_DIS
LIN {X 0.130,Y -491.713,Z 849.516,A 0.000,B 0.000,C 90.000,E1 272.865} C_DIS
LIN {X -0.155,Y -490.513,Z 849.513,A 0.000,B 0.000,C 90.000,E1 272.407} C_DIS
LIN {X 0.049,Y -488.883,Z 849.511,A 0.000,B 0.000,C 90.000,E1 271.892} C_DIS
LIN {X -0.228,Y -486.736,Z 849.508,A 0.000,B 0.000,C 90.000,E1 271.432} C_DIS
LIN {X -0.041,Y -483.994,Z 849.505,A 0.000,B 0.000,C 90.000,E1 270.917} C_DIS
LIN {X 0.125,Y -480.602,Z 849.502,A 0.000,B 0.000,C 90.000,E1 270.401} C_DIS
LIN {X -0.205,Y -476.483,Z 849.500,A 0.000,B 0.000,C 90.000,E1 269.943} C_DIS
LIN {X -0.076,Y -471.504,Z 849.497,A 0.000,B 0.000,C 90.000,E1 269.427} C_DIS
LIN {X -0.160,Y -468.780,Z 849.495,A 0.000,B 0.000,C 90.000,E1 269.198} C_DIS
LIN {X -0.095,Y -462.729,Z 849.493,A 0.000,B 0.000,C 90.000,E1 268.740} C_DIS
LIN {X 0.000,Y -456.087,Z 849.491,A 0.000,B 0.000,C 90.000,E1 268.339} C_DIS
LIN {X 0.176,Y -448.967,Z 849.489,A 0.000,B 0.000,C 90.000,E1 267.993} C_DIS
LIN {X -0.035,Y -441.507,Z 849.488,A 0.000,B 0.000,C 90.000,E1 267.764} C_DIS
LIN {X -0.207,Y -433.406,Z 849.486,A 0.000,B 0.000,C 90.000,E1 267.593} C_DIS
LIN {X 0.031,Y -424.469,Z 849.486,A 0.000,B 0.000,C 90.000,E1 267.421} C_DIS
LIN {X 0.034,Y -418.746,Z 849.485,A 0.000,B 0.000,C 90.000,E1 267.364} C_DIS
LIN {X -0.104,Y -414.202,Z 849.485,A 0.000,B 0.000,C 90.000,E1 267.364} C_DIS
LIN {X -0.076,Y -181.030,Z 849.485,A 0.000,B 0.000,C 90.000,E1 267.364} C_DIS
LIN {X -0.051,Y -180.792,Z 849.471,A 0.000,B 0.000,C 90.000,E1 264.780} C_DIS
LIN {X 0.023,Y -178.890,Z 849.443,A 0.000,B 0.000,C 90.000,E1 259.690} C_DIS
LIN {X -0.071,Y -175.933,Z 849.414,A 0.000,B 0.000,C 90.000,E1 254.629} C_DIS
LIN {X 0.044,Y -175.380,Z 849.410,A 0.000,B 0.000,C 90.000,E1 253.740} C_DIS
LIN {X 0.041,Y -172.154,Z 849.386,A 0.000,B 0.000,C 90.000,E1 249.464} C_DIS
LIN {X 0.079,Y -171.620,Z 849.381,A 0.000,B 0.000,C 90.000,E1 248.592} C_DIS
LIN {X 0.066,Y -167.842,Z 849.357,A 0.000,B 0.000,C 90.000,E1 244.280} C_DIS
LIN {X 0.006,Y -166.572,Z 849.348,A 0.000,B 0.000,C 90.000,E1 242.564} C_DIS
LIN {X -0.007,Y -162.564,Z 849.323,A 0.000,B 0.000,C 90.000,E1 238.201} C_DIS
LIN {X 0.052,Y -161.245,Z 849.314,A 0.000,B 0.000,C 90.000,E1 236.421} C_DIS
LIN {X -0.037,Y -157.248,Z 849.289,A 0.000,B 0.000,C 90.000,E1 232.029} C_DIS
LIN {X 0.010,Y -155.971,Z 849.279,A 0.000,B 0.000,C 90.000,E1 230.231} C_DIS
LIN {X 0.067,Y -152.226,Z 849.254,A 0.000,B 0.000,C 90.000,E1 225.729} C_DIS
LIN {X -0.022,Y -150.468,Z 849.239,A 0.000,B 0.000,C 90.000,E1 223.056} C_DIS
LIN {X -0.002,Y -147.193,Z 849.214,A 0.000,B 0.000,C 90.000,E1 218.508} C_DIS
LIN {X 0.079,Y -145.212,Z 849.194,A 0.000,B 0.000,C 90.000,E1 214.818} C_DIS
LIN {X -0.011,Y -142.345,Z 849.163,A 0.000,B 0.000,C 90.000,E1 209.333} C_DIS
LIN {X 0.043,Y -141.733,Z 849.153,A 0.000,B 0.000,C 90.000,E1 207.462} C_DIS
LIN {X 0.024,Y -139.483,Z 849.117,A 0.000,B 0.000,C 90.000,E1 200.972} C_DIS
LIN {X 0.012,Y -138.984,Z 849.101,A 0.000,B 0.000,C 90.000,E1 198.181} C_DIS
LIN {X -0.026,Y -138.333,Z 849.054,A 0.000,B 0.000,C 90.000,E1 189.792} C_DIS
LIN {X -0.002,Y -139.425,Z 849.008,A 0.000,B 0.000,C 90.000,E1 181.375} C_DIS
LIN {X 0.052,Y -141.349,Z 848.971,A 0.000,B 0.000,C 90.000,E1 174.837} C_DIS
LIN {X 0.029,Y -142.704,Z 848.956,A 0.000,B 0.000,C 90.000,E1 172.064} C_DIS
LIN {X -0.012,Y -145.074,Z 848.930,A 0.000,B 0.000,C 90.000,E1 167.465} C_DIS
LIN {X -0.016,Y -147.699,Z 848.910,A 0.000,B 0.000,C 90.000,E1 163.795} C_DIS
LIN {X 0.017,Y -150.350,Z 848.890,A 0.000,B 0.000,C 90.000,E1 160.134} C_DIS
LIN {X 0.010,Y -154.605,Z 848.865,A 0.000,B 0.000,C 90.000,E1 155.613} C_DIS
LIN {X 0.017,Y -158.147,Z 848.845,A 0.000,B 0.000,C 90.000,E1 152.025} C_DIS
LIN {X 0.061,Y -162.433,Z 848.825,A 0.000,B 0.000,C 90.000,E1 148.456} C_DIS
LIN {X -0.043,Y -166.692,Z 848.805,A 0.000,B 0.000,C 90.000,E1 144.975} C_DIS
LIN {X 0.071,Y -171.698,Z 848.786,A 0.000,B 0.000,C 90.000,E1 141.457} C_DIS
LIN {X 0.005,Y -176.670,Z 848.767,A 0.000,B 0.000,C 90.000,E1 138.038} C_DIS
LIN {X 0.000,Y -180.966,Z 848.753,A 0.000,B 0.000,C 90.000,E1 135.486} C_DIS
LIN {X -0.013,Y -186.391,Z 848.734,A 0.000,B 0.000,C 90.000,E1 132.123} C_DIS
LIN {X -0.073,Y -191.020,Z 848.720,A 0.000,B 0.000,C 90.000,E1 129.644} C_DIS
LIN {X -0.039,Y -192.961,Z 848.714,A 0.000,B 0.000,C 90.000,E1 128.463} C_DIS
LIN {X -0.095,Y -293.746,Z 848.714,A 0.000,B 0.000,C 90.000,E1 128.463} C_DIS
LIN {X 0.077,Y -296.135,Z 848.713,A 0.000,B 0.000,C 90.000,E1 128.382} C_DIS
LIN {X 0.042,Y -300.231,Z 848.712,A 0.000,B 0.000,C 90.000,E1 128.177} C_DIS
LIN {X 0.007,Y -302.641,Z 848.711,A 0.000,B 0.000,C 90.000,E1 127.971} C_DIS
LIN {X 0.087,Y -306.456,Z 848.708,A 0.000,B 0.000,C 90.000,E1 127.443} C_DIS
LIN {X -0.142,Y -308.157,Z 848.706,A 0.000,B 0.000,C 90.000,E1 127.156} C_DIS
LIN {X 0.059,Y -309.489,Z 848.704,A 0.000,B 0.000,C 90.000,E1 126.790} C_DIS
LIN {X 0.052,Y -321.702,Z 848.683,A 0.000,B 0.000,C 90.000,E1 122.911} C_DIS
LIN {X -0.057,Y -332.239,Z 848.667,A 0.000,B 0.000,C 90.000,E1 120.079} C_DIS
LIN {X 0.079,Y -344.140,Z 848.651,A 0.000,B 0.000,C 90.000,E1 117.257} C_DIS
LIN {X 0.087,Y -357.503,Z 848.636,A 0.000,B 0.000,C 90.000,E1 114.515} C_DIS
LIN {X -0.059,Y -370.711,Z 848.623,A 0.000,B 0.000,C 90.000,E1 112.153} C_DIS
LIN {X -0.015,Y -385.264,Z 848.610,A 0.000,B 0.000,C 90.000,E1 109.812} C_DIS
LIN {X 0.128,Y -401.269,Z 848.597,A 0.000,B 0.000,C 90.000,E1 107.511} C_DIS
LIN {X 0.044,Y -418.840,Z 848.585,A 0.000,B 0.000,C 90.000,E1 105.300} C_DIS
LIN {X 0.203,Y -438.070,Z 848.573,A 0.000,B 0.000,C 90.000,E1 103.119} C_DIS
LIN {X 0.000,Y -458.235,Z 848.562,A 0.000,B 0.000,C 90.000,E1 101.130} C_DIS
LIN {X -0.094,Y -468.350,Z 848.557,A 0.000,B 0.000,C 90.000,E1 100.197} C_DIS
LIN {X -0.057,Y -470.176,Z 848.555,A 0.000,B 0.000,C 90.000,E1 99.962} C_DIS
LIN {X -0.207,Y -471.699,Z 848.554,A 0.000,B 0.000,C 90.000,E1 99.726} C_DIS
LIN {X 0.030,Y -472.838,Z 848.552,A 0.000,B 0.000,C 90.000,E1 99.443} C_DIS
LIN {X 0.214,Y -474.203,Z 848.550,A 0.000,B 0.000,C 90.000,E1 98.916} C_DIS
LIN {X -0.138,Y -474.547,Z 848.547,A 0.000,B 0.000,C 90.000,E1 98.454} C_DIS
LIN {X -0.011,Y -473.929,Z 848.544,A 0.000,B 0.000,C 90.000,E1 97.936} C_DIS
LIN {X 0.180,Y -472.251,Z 848.541,A 0.000,B 0.000,C 90.000,E1 97.409} C_DIS
LIN {X -0.023,Y -470.923,Z 848.540,A 0.000,B 0.000,C 90.000,E1 97.182} C_DIS
